LIN {X 0,Y 196.3,Z 471.05,A -85,B 0,C 180,E1 -25408.972,E2 -25408.972} C_VEL
LIN {X 0,Y 193.786,Z 486.083,A -85,B 0,C 180,E1 -25409.629,E2 -25409.629} C_VEL
LIN {X 0,Y 190.214,Z 500.774,A -85,B 0,C 180,E1 -25410.535,E2 -25410.535} C_VEL
LIN {X 0,Y 185.876,Z 514.562,A -85,B 0,C 180,E1 -25411.712,E2 -25411.712} C_VEL
LIN {X 0,Y 180.555,Z 528.47,A -85,B 0,C 180,E1 -25413.314,E2 -25413.314} C_VEL
LIN {X 0,Y 174.309,Z 541.829,A -85,B 0,C 180,E1 -25415.27,E2 -25415.27} C_VEL
LIN {X 0,Y 167.482,Z 554.228,A -85,B 0,C 180,E1 -25417.625,E2 -25417.625} C_VEL
LIN {X 0,Y 160.938,Z 564.609,A -85,B 0,C 180,E1 -25420.166,E2 -25420.166} C_VEL
LIN {X 0,Y 154.161,Z 574.239,A -85,B 0,C 180,E1 -25423.164,E2 -25423.164} C_VEL
LIN {X 0,Y 148.078,Z 582.443,A -85,B 0,C 180,E1 -25426.515,E2 -25426.515} C_VEL
LIN {X 0,Y 141.347,Z 590.516,A -85,B 0,C 180,E1 -25430.659,E2 -25430.659} C_VEL
LIN {X 0,Y 135.368,Z 597.175,A -85,B 0,C 180,E1 -25435.175,E2 -25435.175} C_VEL
LIN {X 0,Y 129.686,Z 603.328,A -85,B 0,C 180,E1 -25440.809,E2 -25440.809} C_VEL
LIN {X 0,Y 125.219,Z 608.071,A -85,B 0,C 180,E1 -25446.867,E2 -25446.867} C_VEL
LIN {X 0,Y 122.097,Z 611.536,A -85,B 0,C 180,E1 -25453.274,E2 -25453.274} C_VEL
LIN {X 0,Y 120.197,Z 613.818,A -85,B 0,C 180,E1 -25459.898,E2 -25459.898} C_VEL
LIN {X 0,Y 119.437,Z 614.974,A -85,B 0,C 180,E1 -25466.627,E2 -25466.627} C_VEL
LIN {X 0,Y 119.419,Z 615.126,A -85,B 0,C 180,E1 -25470,E2 -25470} C_VEL
LIN {X 0,Y 119.683,Z 614.566,A -85,B 0,C 180,E1 -25476.744,E2 -25476.744} C_VEL
LIN {X 0,Y 120.982,Z 612.894,A -85,B 0,C 180,E1 -25483.436,E2 -25483.436} C_VEL
LIN {X 0,Y 123.4,Z 610.069,A -85,B 0,C 180,E1 -25489.981,E2 -25489.981} C_VEL
LIN {X 0,Y 127.319,Z 606.012,A -85,B 0,C 180,E1 -25496.205,E2 -25496.205} C_VEL
LIN {X 0,Y 132.367,Z 600.63,A -85,B 0,C 180,E1 -25502.068,E2 -25502.068} C_VEL
LIN {X 0,Y 138.615,Z 593.765,A -85,B 0,C 180,E1 -25507.474,E2 -25507.474} C_VEL
LIN {X 0,Y 145.953,Z 585.189,A -85,B 0,C 180,E1 -25512.386,E2 -25512.386} C_VEL
LIN {X 0,Y 150.8,Z 579.119,A -85,B 0,C 180,E1 -25515.081,E2 -25515.081} C_VEL
LIN {X 0,Y 156.318,Z 571.624,A -85,B 0,C 180,E1 -25517.886,E2 -25517.886} C_VEL
LIN {X 0,Y 163.24,Z 561.484,A -85,B 0,C 180,E1 -25520.799,E2 -25520.799} C_VEL
LIN {X 0,Y 170.453,Z 549.406,A -85,B 0,C 180,E1 -25523.512,E2 -25523.512} C_VEL
LIN {X 0,Y 176.765,Z 537.285,A -85,B 0,C 180,E1 -25525.586,E2 -25525.586} C_VEL
LIN {X 0,Y 182.653,Z 523.835,A -85,B 0,C 180,E1 -25527.406,E2 -25527.406} C_VEL
LIN {X 0,Y 187.121,Z 511.539,A -85,B 0,C 180,E1 -25528.697,E2 -25528.697} C_VEL
LIN {X 0,Y 191.471,Z 496.805,A -85,B 0,C 180,E1 -25529.865,E2 -25529.865} C_VEL
LIN {X 0,Y 194.807,Z 481.709,A -85,B 0,C 180,E1 -25530.722,E2 -25530.722} C_VEL
LIN {X 0,Y 197.091,Z 466.466,A -85,B 0,C 180,E1 -25531.281,E2 -25531.281} C_VEL
LIN {X 0,Y 201.447,Z 418.406,A -85,B 0,C 180,E1 -25532.593,E2 -25532.593} C_VEL
LIN {X 0,Y 197.597,Z 410.359,A -85,B 0,C 180,E1 -25535.536,E2 -25535.536} C_VEL
LIN {X 0,Y 193.811,Z 403.079,A -85,B 0,C 180,E1 -25538.878,E2 -25538.878} C_VEL
LIN {X 0,Y 190.348,Z 396.957,A -85,B 0,C 180,E1 -25542.543,E2 -25542.543} C_VEL
LIN {X 0,Y 187.688,Z 392.59,A -85,B 0,C 180,E1 -25546.051,E2 -25546.051} C_VEL
LIN {X 0,Y 185.737,Z 388.987,A -85,B 0,C 180,E1 -25549.508,E2 -25549.508} C_VEL
LIN {X 0,Y 183.95,Z 386.282,A -85,B 0,C 180,E1 -25554.207,E2 -25554.207} C_VEL
LIN {X 0,Y 183.494,Z 384.314,A -85,B 0,C 180,E1 -25557.256,E2 -25557.256} C_VEL
LIN {X 0,Y 183.527,Z 384.307,A -85,B 0,C 180,E1 -25562.606,E2 -25562.606} C_VEL
LIN {X 0,Y 185.177,Z 388.442,A -85,B 0,C 180,E1 -25569.007,E2 -25569.007} C_VEL
LIN {X 0,Y 185.895,Z 389.445,A -85,B 0,C 180,E1 -25570.494,E2 -25570.494} C_VEL
LIN {X 0,Y 188.515,Z 393.956,A -85,B 0,C 180,E1 -25574.782,E2 -25574.782} C_VEL
LIN {X 0,Y 190.911,Z 398.053,A -85,B 0,C 180,E1 -25577.767,E2 -25577.767} C_VEL
LIN {X 0,Y 193.357,Z 402.379,A -85,B 0,C 180,E1 -25580.339,E2 -25580.339} C_VEL
LIN {X 0,Y 195.257,Z 406.102,A -85,B 0,C 180,E1 -25582.136,E2 -25582.136} C_VEL
LIN {X 0,Y 198.42,Z 414.111,A -85,B 0,C 180,E1 -25584.943,E2 -25584.943} C_VEL
LIN {X 0,Y 201.237,Z 421.993,A -85,B 0,C 180,E1 -25587.208,E2 -25587.208} C_VEL
LIN {X 0,Y 196.16,Z 476.141,A -85,B 0,C 180,E1 -25588.658,E2 -25588.658} C_VEL
LIN {X 0,Y 193.378,Z 491.918,A -85,B 0,C 180,E1 -25589.283,E2 -25589.283} C_VEL
LIN {X 0,Y 189.569,Z 507.14,A -85,B 0,C 180,E1 -25590.203,E2 -25590.203} C_VEL
LIN {X 0,Y 185.034,Z 520.859,A -85,B 0,C 180,E1 -25591.287,E2 -25591.287} C_VEL
LIN {X 0,Y 179.64,Z 534.306,A -85,B 0,C 180,E1 -25592.742,E2 -25592.742} C_VEL
LIN {X 0,Y 173.552,Z 547.041,A -85,B 0,C 180,E1 -25594.536,E2 -25594.536} C_VEL
LIN {X 0,Y 166.783,Z 559.341,A -85,B 0,C 180,E1 -25596.812,E2 -25596.812} C_VEL
LIN {X 0,Y 159.471,Z 570.819,A -85,B 0,C 180,E1 -25599.537,E2 -25599.537} C_VEL
LIN {X 0,Y 152.629,Z 580.487,A -85,B 0,C 180,E1 -25602.547,E2 -25602.547} C_VEL
LIN {X 0,Y 145.168,Z 590.115,A -85,B 0,C 180,E1 -25606.477,E2 -25606.477} C_VEL
LIN {X 0,Y 138.116,Z 598.719,A -85,B 0,C 180,E1 -25611.243,E2 -25611.243} C_VEL
LIN {X 0,Y 132.184,Z 605.322,A -85,B 0,C 180,E1 -25616.065,E2 -25616.065} C_VEL
LIN {X 0,Y 126.669,Z 611.479,A -85,B 0,C 180,E1 -25622.252,E2 -25622.252} C_VEL
LIN {X 0,Y 124.332,Z 613.407,A -85,B 0,C 180,E1 -25624.578,E2 -25624.578} C_VEL
LIN {X 0,Y 119.213,Z 616.082,A -85,B 0,C 180,E1 -25628.377,E2 -25628.377} C_VEL
LIN {X 0,Y 115.378,Z 617.848,A -85,B 0,C 180,E1 -25631.671,E2 -25631.671} C_VEL
LIN {X 0,Y 113.504,Z 618.991,A -85,B 0,C 180,E1 -25634.42,E2 -25634.42} C_VEL
LIN {X 0,Y 113.194,Z 619.293,A -85,B 0,C 180,E1 -25635.386,E2 -25635.386} C_VEL
LIN {X 0,Y 112.135,Z 621.139,A -85,B 0,C 180,E1 -25642.799,E2 -25642.799} C_VEL
LIN {X 0,Y 112.248,Z 621.75,A -85,B 0,C 180,E1 -25650,E2 -25650} C_VEL
LIN {X 0,Y 112.127,Z 621.12,A -85,B 0,C 180,E1 -25657.201,E2 -25657.201} C_VEL
LIN {X 0,Y 113.113,Z 619.332,A -85,B 0,C 180,E1 -25664.39,E2 -25664.39} C_VEL
LIN {X 0,Y 115.543,Z 616.373,A -85,B 0,C 180,E1 -25671.404,E2 -25671.404} C_VEL
LIN {X 0,Y 119.342,Z 612.172,A -85,B 0,C 180,E1 -25678.106,E2 -25678.106} C_VEL
LIN {X 0,Y 124.758,Z 606.631,A -85,B 0,C 180,E1 -25684.285,E2 -25684.285} C_VEL
LIN {X 0,Y 131.502,Z 599.596,A -85,B 0,C 180,E1 -25689.89,E2 -25689.89} C_VEL
LIN {X 0,Y 138.345,Z 591.848,A -85,B 0,C 180,E1 -25694.499,E2 -25694.499} C_VEL
LIN {X 0,Y 145.593,Z 583.013,A -85,B 0,C 180,E1 -25698.433,E2 -25698.433} C_VEL
LIN {X 0,Y 153.801,Z 572.132,A -85,B 0,C 180,E1 -25702.02,E2 -25702.02} C_VEL
LIN {X 0,Y 161.305,Z 560.935,A -85,B 0,C 180,E1 -25704.777,E2 -25704.777} C_VEL
LIN {X 0,Y 168.449,Z 548.675,A -85,B 0,C 180,E1 -25707.096,E2 -25707.096} C_VEL
LIN {X 0,Y 175.181,Z 535.171,A -85,B 0,C 180,E1 -25709.038,E2 -25709.038} C_VEL
LIN {X 0,Y 180.74,Z 521.912,A -85,B 0,C 180,E1 -25710.46,E2 -25710.46} C_VEL
LIN {X 0,Y 185.715,Z 507.4,A -85,B 0,C 180,E1 -25711.621,E2 -25711.621} C_VEL
LIN {X 0,Y 189.648,Z 492.344,A -85,B 0,C 180,E1 -25712.505,E2 -25712.505} C_VEL
LIN {X 0,Y 192.467,Z 477.05,A -85,B 0,C 180,E1 -25713.108,E2 -25713.108} C_VEL
LIN {X 0,Y 195.922,Z 442.724,A -85,B 0,C 180,E1 -25714.03,E2 -25714.03} C_VEL
LIN {X 0,Y 197.57,Z 424.787,A -85,B 0,C 180,E1 -25714.509,E2 -25714.509} C_VEL
LIN {X 0,Y 194.282,Z 415.387,A -85,B 0,C 180,E1 -25717.467,E2 -25717.467} C_VEL
LIN {X 0,Y 191.942,Z 409.582,A -85,B 0,C 180,E1 -25719.796,E2 -25719.796} C_VEL
LIN {X 0,Y 188.507,Z 403.239,A -85,B 0,C 180,E1 -25723.624,E2 -25723.624} C_VEL
LIN {X 0,Y 186.244,Z 399.273,A -85,B 0,C 180,E1 -25726.776,E2 -25726.776} C_VEL
LIN {X 0,Y 184.295,Z 395.581,A -85,B 0,C 180,E1 -25730.396,E2 -25730.396} C_VEL
LIN {X 0,Y 182.635,Z 392.54,A -85,B 0,C 180,E1 -25735.31,E2 -25735.31} C_VEL
LIN {X 0,Y 182.364,Z 391.3,A -85,B 0,C 180,E1 -25737.239,E2 -25737.239} C_VEL
LIN {X 0,Y 182.151,Z 391.03,A -85,B 0,C 180,E1 -25740,E2 -25740} C_VEL
LIN {X 0,Y 182.429,Z 391.531,A -85,B 0,C 180,E1 -25743.728,E2 -25743.728} C_VEL
LIN {X 0,Y 183.828,Z 395.187,A -85,B 0,C 180,E1 -25749.074,E2 -25749.074} C_VEL
LIN {X 0,Y 184.521,Z 396.112,A -85,B 0,C 180,E1 -25750.562,E2 -25750.562} C_VEL
LIN {X 0,Y 186.923,Z 400.501,A -85,B 0,C 180,E1 -25754.702,E2 -25754.702} C_VEL
LIN {X 0,Y 189.266,Z 404.677,A -85,B 0,C 180,E1 -25757.756,E2 -25757.756} C_VEL
LIN {X 0,Y 192.494,Z 410.713,A -85,B 0,C 180,E1 -25761.204,E2 -25761.204} C_VEL
LIN {X 0,Y 195.769,Z 417.37,A -85,B 0,C 180,E1 -25764.172,E2 -25764.172} C_VEL
LIN {X 0,Y 197.776,Z 421.755,A -85,B 0,C 180,E1 -25765.813,E2 -25765.813} C_VEL
LIN {X 0,Y 193.089,Z 470.398,A -85,B 0,C 180,E1 -25767.1,E2 -25767.1} C_VEL
LIN {X 0,Y 190.382,Z 486.296,A -85,B 0,C 180,E1 -25767.775,E2 -25767.775} C_VEL
LIN {X 0,Y 186.708,Z 500.985,A -85,B 0,C 180,E1 -25768.658,E2 -25768.658} C_VEL
LIN {X 0,Y 182.243,Z 514.772,A -85,B 0,C 180,E1 -25769.812,E2 -25769.812} C_VEL
LIN {X 0,Y 176.917,Z 528.235,A -85,B 0,C 180,E1 -25771.322,E2 -25771.322} C_VEL
LIN {X 0,Y 170.981,Z 540.748,A -85,B 0,C 180,E1 -25773.126,E2 -25773.126} C_VEL
LIN {X 0,Y 164.496,Z 552.307,A -85,B 0,C 180,E1 -25775.207,E2 -25775.207} C_VEL
LIN {X 0,Y 157.704,Z 563.04,A -85,B 0,C 180,E1 -25777.721,E2 -25777.721} C_VEL
LIN {X 0,Y 150.543,Z 572.967,A -85,B 0,C 180,E1 -25780.659,E2 -25780.659} C_VEL
LIN {X 0,Y 143.006,Z 582.648,A -85,B 0,C 180,E1 -25784.555,E2 -25784.555} C_VEL
LIN {X 0,Y 135.9,Z 590.722,A -85,B 0,C 180,E1 -25788.75,E2 -25788.75} C_VEL
LIN {X 0,Y 129.57,Z 597.381,A -85,B 0,C 180,E1 -25793.371,E2 -25793.371} C_VEL
LIN {X 0,Y 123.508,Z 603.533,A -85,B 0,C 180,E1 -25799.195,E2 -25799.195} C_VEL
LIN {X 0,Y 118.713,Z 608.276,A -85,B 0,C 180,E1 -25805.518,E2 -25805.518} C_VEL
LIN {X 0,Y 115.272,Z 611.741,A -85,B 0,C 180,E1 -25812.252,E2 -25812.252} C_VEL
LIN {X 0,Y 113.203,Z 614.022,A -85,B 0,C 180,E1 -25819.266,E2 -25819.266} C_VEL
LIN {X 0,Y 112.353,Z 615.177,A -85,B 0,C 180,E1 -25826.414,E2 -25826.414} C_VEL
LIN {X 0,Y 112.335,Z 615.329,A -85,B 0,C 180,E1 -25830,E2 -25830} C_VEL
LIN {X 0,Y 112.624,Z 614.769,A -85,B 0,C 180,E1 -25837.169,E2 -25837.169} C_VEL
LIN {X 0,Y 114.05,Z 613.098,A -85,B 0,C 180,E1 -25844.269,E2 -25844.269} C_VEL
LIN {X 0,Y 116.717,Z 610.273,A -85,B 0,C 180,E1 -25851.178,E2 -25851.178} C_VEL
LIN {X 0,Y 120.945,Z 606.215,A -85,B 0,C 180,E1 -25857.701,E2 -25857.701} C_VEL
LIN {X 0,Y 126.368,Z 600.833,A -85,B 0,C 180,E1 -25863.789,E2 -25863.789} C_VEL
LIN {X 0,Y 133.009,Z 593.968,A -85,B 0,C 180,E1 -25869.349,E2 -25869.349} C_VEL
LIN {X 0,Y 140.792,Z 585.39,A -85,B 0,C 180,E1 -25874.333,E2 -25874.333} C_VEL
LIN {X 0,Y 146.284,Z 578.73,A -85,B 0,C 180,E1 -25877.329,E2 -25877.329} C_VEL
LIN {X 0,Y 152.796,Z 570.211,A -85,B 0,C 180,E1 -25880.391,E2 -25880.391} C_VEL
LIN {X 0,Y 160.079,Z 559.807,A -85,B 0,C 180,E1 -25883.246,E2 -25883.246} C_VEL
LIN {X 0,Y 166.963,Z 548.488,A -85,B 0,C 180,E1 -25885.695,E2 -25885.695} C_VEL
LIN {X 0,Y 173.517,Z 536.181,A -85,B 0,C 180,E1 -25887.724,E2 -25887.724} C_VEL
LIN {X 0,Y 179.503,Z 522.719,A -85,B 0,C 180,E1 -25889.467,E2 -25889.467} C_VEL
LIN {X 0,Y 184.555,Z 508.759,A -85,B 0,C 180,E1 -25890.862,E2 -25890.862} C_VEL
LIN {X 0,Y 188.693,Z 494.404,A -85,B 0,C 180,E1 -25891.913,E2 -25891.913} C_VEL
LIN {X 0,Y 192.06,Z 478.698,A -85,B 0,C 180,E1 -25892.714,E2 -25892.714} C_VEL
LIN {X 0,Y 194.184,Z 463.277,A -85,B 0,C 180,E1 -25893.208,E2 -25893.208} C_VEL
LIN {X 0,Y 198.031,Z 421.974,A -85,B 0,C 180,E1 -25894.285,E2 -25894.285} C_VEL
LIN {X 0,Y 194.199,Z 413.869,A -85,B 0,C 180,E1 -25897.526,E2 -25897.526} C_VEL
LIN {X 0,Y 190.907,Z 407.427,A -85,B 0,C 180,E1 -25900.79,E2 -25900.79} C_VEL
LIN {X 0,Y 188.19,Z 402.537,A -85,B 0,C 180,E1 -25904.013,E2 -25904.013} C_VEL
LIN {X 0,Y 186.384,Z 399.332,A -85,B 0,C 180,E1 -25906.63,E2 -25906.63} C_VEL
LIN {X 0,Y 184.403,Z 395.666,A -85,B 0,C 180,E1 -25910.401,E2 -25910.401} C_VEL
LIN {X 0,Y 182.769,Z 392.393,A -85,B 0,C 180,E1 -25915.796,E2 -25915.796} C_VEL
LIN {X 0,Y 182.625,Z 391.396,A -85,B 0,C 180,E1 -25917.243,E2 -25917.243} C_VEL
LIN {X 0,Y 182.608,Z 391.312,A -85,B 0,C 180,E1 -25922.205,E2 -25922.205} C_VEL
LIN {X 0,Y 184.439,Z 395.708,A -85,B 0,C 180,E1 -25929.32,E2 -25929.32} C_VEL
LIN {X 0,Y 187.113,Z 400.621,A -85,B 0,C 180,E1 -25934.131,E2 -25934.131} C_VEL
LIN {X 0,Y 189.335,Z 404.558,A -85,B 0,C 180,E1 -25937.066,E2 -25937.066} C_VEL
LIN {X 0,Y 192.506,Z 410.448,A -85,B 0,C 180,E1 -25940.502,E2 -25940.502} C_VEL
LIN {X 0,Y 195.434,Z 418.137,A -85,B 0,C 180,E1 -25943.371,E2 -25943.371} C_VEL
LIN {X 0,Y 197.796,Z 425.06,A -85,B 0,C 180,E1 -25945.469,E2 -25945.469} C_VEL
LIN {X 0,Y 192.822,Z 476.142,A -85,B 0,C 180,E1 -25946.81,E2 -25946.81} C_VEL
LIN {X 0,Y 190.008,Z 491.724,A -85,B 0,C 180,E1 -25947.416,E2 -25947.416} C_VEL
LIN {X 0,Y 186.079,Z 506.942,A -85,B 0,C 180,E1 -25948.302,E2 -25948.302} C_VEL
LIN {X 0,Y 181.444,Z 520.662,A -85,B 0,C 180,E1 -25949.368,E2 -25949.368} C_VEL
LIN {X 0,Y 175.9,Z 534.108,A -85,B 0,C 180,E1 -25950.796,E2 -25950.796} C_VEL
LIN {X 0,Y 169.641,Z 546.794,A -85,B 0,C 180,E1 -25952.547,E2 -25952.547} C_VEL
LIN {X 0,Y 162.618,Z 559.141,A -85,B 0,C 180,E1 -25954.803,E2 -25954.803} C_VEL
LIN {X 0,Y 155.01,Z 570.617,A -85,B 0,C 180,E1 -25957.495,E2 -25957.495} C_VEL
LIN {X 0,Y 147.888,Z 580.285,A -85,B 0,C 180,E1 -25960.506,E2 -25960.506} C_VEL
LIN {X 0,Y 140.157,Z 589.787,A -85,B 0,C 180,E1 -25964.396,E2 -25964.396} C_VEL
LIN {X 0,Y 133.324,Z 597.716,A -85,B 0,C 180,E1 -25968.784,E2 -25968.784} C_VEL
LIN {X 0,Y 126.283,Z 605.118,A -85,B 0,C 180,E1 -25974.244,E2 -25974.244} C_VEL
LIN {X 0,Y 120.625,Z 611.002,A -85,B 0,C 180,E1 -25980.315,E2 -25980.315} C_VEL
LIN {X 0,Y 117.351,Z 614.51,A -85,B 0,C 180,E1 -25985.215,E2 -25985.215} C_VEL
LIN {X 0,Y 114.117,Z 618.057,A -85,B 0,C 180,E1 -25992.066,E2 -25992.066} C_VEL
LIN {X 0,Y 113.194,Z 619.293,A -85,B 0,C 180,E1 -25995.386,E2 -25995.386} C_VEL
LIN {X 0,Y 112.042,Z 620.233,A -85,B 0,C 180,E1 -25998.29,E2 -25998.29} C_VEL
LIN {X 0,Y 110.209,Z 620.902,A -85,B 0,C 180,E1 -26001.18,E2 -26001.18} C_VEL
LIN {X 0,Y 106.313,Z 621.518,A -85,B 0,C 180,E1 -26007.182,E2 -26007.182} C_VEL
LIN {X 0,Y 105.049,Z 621.484,A -85,B 0,C 180,E1 -26011.468,E2 -26011.468} C_VEL
LIN {X 0,Y 105.054,Z 620.915,A -85,B 0,C 180,E1 -26017.689,E2 -26017.689} C_VEL
LIN {X 0,Y 106.195,Z 619.127,A -85,B 0,C 180,E1 -26025.35,E2 -26025.35} C_VEL
LIN {X 0,Y 108.882,Z 616.167,A -85,B 0,C 180,E1 -26032.785,E2 -26032.785} C_VEL
LIN {X 0,Y 113.068,Z 611.966,A -85,B 0,C 180,E1 -26039.818,E2 -26039.818} C_VEL
LIN {X 0,Y 118.897,Z 606.424,A -85,B 0,C 180,E1 -26046.234,E2 -26046.234} C_VEL
LIN {X 0,Y 126.073,Z 599.389,A -85,B 0,C 180,E1 -26051.984,E2 -26051.984} C_VEL
LIN {X 0,Y 134.165,Z 590.637,A -85,B 0,C 180,E1 -26057.168,E2 -26057.168} C_VEL
LIN {X 0,Y 142.145,Z 581.353,A -85,B 0,C 180,E1 -26061.141,E2 -26061.141} C_VEL
LIN {X 0,Y 149.5,Z 571.924,A -85,B 0,C 180,E1 -26064.184,E2 -26064.184} C_VEL
LIN {X 0,Y 157.306,Z 560.729,A -85,B 0,C 180,E1 -26066.895,E2 -26066.895} C_VEL
LIN {X 0,Y 164.799,Z 548.256,A -85,B 0,C 180,E1 -26069.22,E2 -26069.22} C_VEL
LIN {X 0,Y 171.632,Z 534.963,A -85,B 0,C 180,E1 -26071.074,E2 -26071.074} C_VEL
LIN {X 0,Y 177.35,Z 521.704,A -85,B 0,C 180,E1 -26072.455,E2 -26072.455} C_VEL
LIN {X 0,Y 182.449,Z 507.19,A -85,B 0,C 180,E1 -26073.582,E2 -26073.582} C_VEL
LIN {X 0,Y 186.479,Z 492.131,A -85,B 0,C 180,E1 -26074.439,E2 -26074.439} C_VEL
LIN {X 0,Y 189.288,Z 477.3,A -85,B 0,C 180,E1 -26075.008,E2 -26075.008} C_VEL
LIN {X 0,Y 192.26,Z 449.441,A -85,B 0,C 180,E1 -26075.744,E2 -26075.744} C_VEL
LIN {X 0,Y 194.297,Z 427.907,A -85,B 0,C 180,E1 -26076.313,E2 -26076.313} C_VEL
LIN {X 0,Y 191.509,Z 419.557,A -85,B 0,C 180,E1 -26079.105,E2 -26079.105} C_VEL
LIN {X 0,Y 189.918,Z 415.545,A -85,B 0,C 180,E1 -26080.827,E2 -26080.827} C_VEL
LIN {X 0,Y 186.997,Z 409.783,A -85,B 0,C 180,E1 -26084.328,E2 -26084.328} C_VEL
LIN {X 0,Y 184.859,Z 405.856,A -85,B 0,C 180,E1 -26087.513,E2 -26087.513} C_VEL
LIN {X 0,Y 183.045,Z 402.324,A -85,B 0,C 180,E1 -26091.166,E2 -26091.166} C_VEL
LIN {X 0,Y 181.513,Z 398.523,A -85,B 0,C 180,E1 -26097.018,E2 -26097.018} C_VEL
LIN {X 0,Y 181.285,Z 398.078,A -85,B 0,C 180,E1 -26100,E2 -26100} C_VEL
LIN {X 0,Y 181.503,Z 398.469,A -85,B 0,C 180,E1 -26103.33,E2 -26103.33} C_VEL
LIN {X 0,Y 182.735,Z 402.024,A -85,B 0,C 180,E1 -26108.571,E2 -26108.571} C_VEL
LIN {X 0,Y 183.447,Z 403.081,A -85,B 0,C 180,E1 -26110.206,E2 -26110.206} C_VEL
LIN {X 0,Y 185.671,Z 407.394,A -85,B 0,C 180,E1 -26114.243,E2 -26114.243} C_VEL
LIN {X 0,Y 187.833,Z 411.455,A -85,B 0,C 180,E1 -26117.207,E2 -26117.207} C_VEL
LIN {X 0,Y 191.052,Z 417.854,A -85,B 0,C 180,E1 -26120.807,E2 -26120.807} C_VEL
LIN {X 0,Y 193.879,Z 424.017,A -85,B 0,C 180,E1 -26123.5,E2 -26123.5} C_VEL
LIN {X 0,Y 194.477,Z 425.359,A -85,B 0,C 180,E1 -26124.027,E2 -26124.027} C_VEL
LIN {X 0,Y 189.877,Z 471.308,A -85,B 0,C 180,E1 -26125.226,E2 -26125.226} C_VEL
LIN {X 0,Y 187.181,Z 486.509,A -85,B 0,C 180,E1 -26125.853,E2 -26125.853} C_VEL
LIN {X 0,Y 183.418,Z 501.195,A -85,B 0,C 180,E1 -26126.717,E2 -26126.717} C_VEL
LIN {X 0,Y 178.818,Z 514.981,A -85,B 0,C 180,E1 -26127.837,E2 -26127.837} C_VEL
LIN {X 0,Y 173.1,Z 528.968,A -85,B 0,C 180,E1 -26129.378,E2 -26129.378} C_VEL
LIN {X 0,Y 166.527,Z 542.242,A -85,B 0,C 180,E1 -26131.285,E2 -26131.285} C_VEL
LIN {X 0,Y 159.205,Z 554.641,A -85,B 0,C 180,E1 -26133.571,E2 -26133.571} C_VEL
LIN {X 0,Y 152.165,Z 565.021,A -85,B 0,C 180,E1 -26136.075,E2 -26136.075} C_VEL
LIN {X 0,Y 144.085,Z 575.518,A -85,B 0,C 180,E1 -26139.353,E2 -26139.353} C_VEL
LIN {X 0,Y 136.98,Z 584.077,A -85,B 0,C 180,E1 -26143.021,E2 -26143.021} C_VEL
LIN {X 0,Y 129.619,Z 591.927,A -85,B 0,C 180,E1 -26147.333,E2 -26147.333} C_VEL
LIN {X 0,Y 122.174,Z 599.251,A -85,B 0,C 180,E1 -26152.844,E2 -26152.844} C_VEL
LIN {X 0,Y 115.996,Z 605.051,A -85,B 0,C 180,E1 -26159.003,E2 -26159.003} C_VEL
LIN {X 0,Y 112.276,Z 608.48,A -85,B 0,C 180,E1 -26164.014,E2 -26164.014} C_VEL
LIN {X 0,Y 108.494,Z 611.945,A -85,B 0,C 180,E1 -26171.102,E2 -26171.102} C_VEL
LIN {X 0,Y 106.216,Z 614.226,A -85,B 0,C 180,E1 -26178.551,E2 -26178.551} C_VEL
LIN {X 0,Y 105.265,Z 615.38,A -85,B 0,C 180,E1 -26186.172,E2 -26186.172} C_VEL
LIN {X 0,Y 105.237,Z 615.532,A -85,B 0,C 180,E1 -26190,E2 -26190} C_VEL
LIN {X 0,Y 105.592,Z 614.972,A -85,B 0,C 180,E1 -26197.649,E2 -26197.649} C_VEL
LIN {X 0,Y 107.157,Z 613.301,A -85,B 0,C 180,E1 -26205.209,E2 -26205.209} C_VEL
LIN {X 0,Y 110.093,Z 610.476,A -85,B 0,C 180,E1 -26212.52,E2 -26212.52} C_VEL
LIN {X 0,Y 114.654,Z 606.419,A -85,B 0,C 180,E1 -26219.365,E2 -26219.365} C_VEL
LIN {X 0,Y 120.496,Z 601.036,A -85,B 0,C 180,E1 -26225.679,E2 -26225.679} C_VEL
LIN {X 0,Y 127.579,Z 594.17,A -85,B 0,C 180,E1 -26231.379,E2 -26231.379} C_VEL
LIN {X 0,Y 134.676,Z 586.787,A -85,B 0,C 180,E1 -26235.85,E2 -26235.85} C_VEL
LIN {X 0,Y 140.198,Z 580.569,A -85,B 0,C 180,E1 -26238.756,E2 -26238.756} C_VEL
LIN {X 0,Y 145.939,Z 573.518,A -85,B 0,C 180,E1 -26241.493,E2 -26241.493} C_VEL
LIN {X 0,Y 153.364,Z 563.66,A -85,B 0,C 180,E1 -26244.428,E2 -26244.428} C_VEL
LIN {X 0,Y 161.08,Z 551.935,A -85,B 0,C 180,E1 -26247.126,E2 -26247.126} C_VEL
LIN {X 0,Y 168.464,Z 538.969,A -85,B 0,C 180,E1 -26249.363,E2 -26249.363} C_VEL
LIN {X 0,Y 174.776,Z 525.676,A -85,B 0,C 180,E1 -26251.148,E2 -26251.148} C_VEL
LIN {X 0,Y 180.165,Z 511.931,A -85,B 0,C 180,E1 -26252.551,E2 -26252.551} C_VEL
LIN {X 0,Y 184.765,Z 497.193,A -85,B 0,C 180,E1 -26253.667,E2 -26253.667} C_VEL
LIN {X 0,Y 188.185,Z 482.602,A -85,B 0,C 180,E1 -26254.461,E2 -26254.461} C_VEL
LIN {X 0,Y 190.589,Z 467.616,A -85,B 0,C 180,E1 -26254.999,E2 -26254.999} C_VEL
LIN {X 0,Y 194.71,Z 425.601,A -85,B 0,C 180,E1 -26256.086,E2 -26256.086} C_VEL
LIN {X 0,Y 191.488,Z 418.43,A -85,B 0,C 180,E1 -26259.116,E2 -26259.116} C_VEL
LIN {X 0,Y 188.418,Z 412.32,A -85,B 0,C 180,E1 -26262.498,E2 -26262.498} C_VEL
LIN {X 0,Y 186.278,Z 408.315,A -85,B 0,C 180,E1 -26265.344,E2 -26265.344} C_VEL
LIN {X 0,Y 185.082,Z 406.027,A -85,B 0,C 180,E1 -26267.249,E2 -26267.249} C_VEL
LIN {X 0,Y 183.291,Z 402.526,A -85,B 0,C 180,E1 -26270.899,E2 -26270.899} C_VEL
LIN {X 0,Y 181.794,Z 399.091,A -85,B 0,C 180,E1 -26276.537,E2 -26276.537} C_VEL
LIN {X 0,Y 181.701,Z 398.351,A -85,B 0,C 180,E1 -26277.783,E2 -26277.783} C_VEL
LIN {X 0,Y 181.737,Z 398.416,A -85,B 0,C 180,E1 -26282.216,E2 -26282.216} C_VEL
LIN {X 0,Y 183.207,Z 402.429,A -85,B 0,C 180,E1 -26288.548,E2 -26288.548} C_VEL
LIN {X 0,Y 183.785,Z 403.582,A -85,B 0,C 180,E1 -26289.909,E2 -26289.909} C_VEL
LIN {X 0,Y 185.779,Z 407.347,A -85,B 0,C 180,E1 -26293.537,E2 -26293.537} C_VEL
LIN {X 0,Y 188.053,Z 411.631,A -85,B 0,C 180,E1 -26296.696,E2 -26296.696} C_VEL
LIN {X 0,Y 190.757,Z 417.016,A -85,B 0,C 180,E1 -26299.785,E2 -26299.785} C_VEL
LIN {X 0,Y 193.452,Z 424.761,A -85,B 0,C 180,E1 -26302.616,E2 -26302.616} C_VEL
LIN {X 0,Y 194.519,Z 428.093,A -85,B 0,C 180,E1 -26303.653,E2 -26303.653} C_VEL
LIN {X 0,Y 189.702,Z 476.124,A -85,B 0,C 180,E1 -26304.905,E2 -26304.905} C_VEL
LIN {X 0,Y 186.847,Z 491.531,A -85,B 0,C 180,E1 -26305.484,E2 -26305.484} C_VEL
LIN {X 0,Y 182.811,Z 506.746,A -85,B 0,C 180,E1 -26306.336,E2 -26306.336} C_VEL
LIN {X 0,Y 178.07,Z 520.465,A -85,B 0,C 180,E1 -26307.377,E2 -26307.377} C_VEL
LIN {X 0,Y 172.36,Z 533.909,A -85,B 0,C 180,E1 -26308.76,E2 -26308.76} C_VEL
LIN {X 0,Y 166.058,Z 546.316,A -85,B 0,C 180,E1 -26310.427,E2 -26310.427} C_VEL
LIN {X 0,Y 158.667,Z 558.941,A -85,B 0,C 180,E1 -26312.694,E2 -26312.694} C_VEL
LIN {X 0,Y 150.766,Z 570.416,A -85,B 0,C 180,E1 -26315.339,E2 -26315.339} C_VEL
LIN {X 0,Y 143.336,Z 580.082,A -85,B 0,C 180,E1 -26318.327,E2 -26318.327} C_VEL
LIN {X 0,Y 135.229,Z 589.583,A -85,B 0,C 180,E1 -26322.22,E2 -26322.22} C_VEL
LIN {X 0,Y 128.006,Z 597.512,A -85,B 0,C 180,E1 -26326.664,E2 -26326.664} C_VEL
LIN {X 0,Y 120.537,Z 604.914,A -85,B 0,C 180,E1 -26332.252,E2 -26332.252} C_VEL
LIN {X 0,Y 114.45,Z 610.798,A -85,B 0,C 180,E1 -26338.537,E2 -26338.537} C_VEL
LIN {X 0,Y 110.886,Z 614.306,A -85,B 0,C 180,E1 -26343.663,E2 -26343.663} C_VEL
LIN {X 0,Y 107.331,Z 617.853,A -85,B 0,C 180,E1 -26350.89,E2 -26350.89} C_VEL
LIN {X 0,Y 105.484,Z 620.199,A -85,B 0,C 180,E1 -26358.47,E2 -26358.47} C_VEL
LIN {X 0,Y 105.007,Z 621.387,A -85,B 0,C 180,E1 -26366.162,E2 -26366.162} C_VEL
LIN {X 0,Y 105.166,Z 621.548,A -85,B 0,C 180,E1 -26370,E2 -26370} C_VEL
LIN {X 0,Y 105.049,Z 621.484,A -85,B 0,C 180,E1 -26371.468,E2 -26371.468} C_VEL
LIN {X 0,Y 104.287,Z 621.291,A -85,B 0,C 180,E1 -26374.668,E2 -26374.668} C_VEL
LIN {X 0,Y 101.684,Z 620.469,A -85,B 0,C 180,E1 -26379.978,E2 -26379.978} C_VEL
LIN {X 0,Y 99.934,Z 619.491,A -85,B 0,C 180,E1 -26384.385,E2 -26384.385} C_VEL
LIN {X 0,Y 99.851,Z 618.377,A -85,B 0,C 180,E1 -26388.319,E2 -26388.319} C_VEL
LIN {X 0,Y 100.01,Z 618.119,A -85,B 0,C 180,E1 -26388.872,E2 -26388.872} C_VEL
LIN {X 0,Y 102.292,Z 615.96,A -85,B 0,C 180,E1 -26394.344,E2 -26394.344} C_VEL
LIN {X 0,Y 106.92,Z 611.761,A -85,B 0,C 180,E1 -26401.725,E2 -26401.725} C_VEL
LIN {X 0,Y 113.18,Z 606.218,A -85,B 0,C 180,E1 -26408.385,E2 -26408.385} C_VEL
LIN {X 0,Y 120.843,Z 599.182,A -85,B 0,C 180,E1 -26414.257,E2 -26414.257} C_VEL
LIN {X 0,Y 128.298,Z 591.623,A -85,B 0,C 180,E1 -26418.903,E2 -26418.903} C_VEL
LIN {X 0,Y 136.523,Z 582.599,A -85,B 0,C 180,E1 -26422.929,E2 -26422.929} C_VEL
LIN {X 0,Y 145.435,Z 571.717,A -85,B 0,C 180,E1 -26426.467,E2 -26426.467} C_VEL
LIN {X 0,Y 153.535,Z 560.522,A -85,B 0,C 180,E1 -26429.12,E2 -26429.12} C_VEL
LIN {X 0,Y 160.724,Z 548.951,A -85,B 0,C 180,E1 -26431.25,E2 -26431.25} C_VEL
LIN {X 0,Y 167.578,Z 536.186,A -85,B 0,C 180,E1 -26433.021,E2 -26433.021} C_VEL
LIN {X 0,Y 173.436,Z 523.264,A -85,B 0,C 180,E1 -26434.368,E2 -26434.368} C_VEL
LIN {X 0,Y 178.638,Z 509.238,A -85,B 0,C 180,E1 -26435.472,E2 -26435.472} C_VEL
LIN {X 0,Y 182.957,Z 494.207,A -85,B 0,C 180,E1 -26436.333,E2 -26436.333} C_VEL
LIN {X 0,Y 186.096,Z 478.965,A -85,B 0,C 180,E1 -26436.922,E2 -26436.922} C_VEL
LIN {X 0,Y 188.504,Z 458.616,A -85,B 0,C 180,E1 -26437.483,E2 -26437.483} C_VEL
LIN {X 0,Y 191.212,Z 431.099,A -85,B 0,C 180,E1 -26438.176,E2 -26438.176} C_VEL
LIN {X 0,Y 188.943,Z 423.955,A -85,B 0,C 180,E1 -26440.724,E2 -26440.724} C_VEL
LIN {X 0,Y 187.789,Z 421.09,A -85,B 0,C 180,E1 -26442.086,E2 -26442.086} C_VEL
LIN {X 0,Y 185.232,Z 415.854,A -85,B 0,C 180,E1 -26445.442,E2 -26445.442} C_VEL
LIN {X 0,Y 183.543,Z 412.509,A -85,B 0,C 180,E1 -26448.193,E2 -26448.193} C_VEL
LIN {X 0,Y 181.945,Z 409.173,A -85,B 0,C 180,E1 -26451.672,E2 -26451.672} C_VEL
LIN {X 0,Y 180.564,Z 405.29,A -85,B 0,C 180,E1 -26457.77,E2 -26457.77} C_VEL
LIN {X 0,Y 180.511,Z 405.276,A -85,B 0,C 180,E1 -26462.232,E2 -26462.232} C_VEL
LIN {X 0,Y 180.639,Z 405.925,A -85,B 0,C 180,E1 -26463.625,E2 -26463.625} C_VEL
LIN {X 0,Y 181.987,Z 409.264,A -85,B 0,C 180,E1 -26468.886,E2 -26468.886} C_VEL
LIN {X 0,Y 184.19,Z 413.757,A -85,B 0,C 180,E1 -26473.375,E2 -26473.375} C_VEL
LIN {X 0,Y 186.26,Z 417.896,A -85,B 0,C 180,E1 -26476.439,E2 -26476.439} C_VEL
LIN {X 0,Y 189.168,Z 424.048,A -85,B 0,C 180,E1 -26479.924,E2 -26479.924} C_VEL
LIN {X 0,Y 191.344,Z 429.064,A -85,B 0,C 180,E1 -26482.169,E2 -26482.169} C_VEL
LIN {X 0,Y 186.895,Z 471.959,A -85,B 0,C 180,E1 -26483.275,E2 -26483.275} C_VEL
LIN {X 0,Y 184.205,Z 486.721,A -85,B 0,C 180,E1 -26483.871,E2 -26483.871} C_VEL
LIN {X 0,Y 180.346,Z 501.405,A -85,B 0,C 180,E1 -26484.708,E2 -26484.708} C_VEL
LIN {X 0,Y 175.623,Z 515.19,A -85,B 0,C 180,E1 -26485.793,E2 -26485.793} C_VEL
LIN {X 0,Y 169.531,Z 529.622,A -85,B 0,C 180,E1 -26487.342,E2 -26487.342} C_VEL
LIN {X 0,Y 162.958,Z 542.449,A -85,B 0,C 180,E1 -26489.155,E2 -26489.155} C_VEL
LIN {X 0,Y 155.389,Z 554.848,A -85,B 0,C 180,E1 -26491.388,E2 -26491.388} C_VEL
LIN {X 0,Y 148.1,Z 565.227,A -85,B 0,C 180,E1 -26493.857,E2 -26493.857} C_VEL
LIN {X 0,Y 140.422,Z 574.856,A -85,B 0,C 180,E1 -26496.797,E2 -26496.797} C_VEL
LIN {X 0,Y 132.236,Z 584.282,A -85,B 0,C 180,E1 -26500.771,E2 -26500.771} C_VEL
LIN {X 0,Y 124.463,Z 592.133,A -85,B 0,C 180,E1 -26505.105,E2 -26505.105} C_VEL
LIN {X 0,Y 116.563,Z 599.456,A -85,B 0,C 180,E1 -26510.724,E2 -26510.724} C_VEL
LIN {X 0,Y 109.942,Z 605.256,A -85,B 0,C 180,E1 -26517.088,E2 -26517.088} C_VEL
LIN {X 0,Y 105.91,Z 608.685,A -85,B 0,C 180,E1 -26522.323,E2 -26522.323} C_VEL
LIN {X 0,Y 101.774,Z 612.15,A -85,B 0,C 180,E1 -26529.802,E2 -26529.802} C_VEL
LIN {X 0,Y 99.262,Z 614.429,A -85,B 0,C 180,E1 -26537.737,E2 -26537.737} C_VEL
LIN {X 0,Y 98.189,Z 615.583,A -85,B 0,C 180,E1 -26545.896,E2 -26545.896} C_VEL
LIN {X 0,Y 98.151,Z 615.734,A -85,B 0,C 180,E1 -26550,E2 -26550} C_VEL
LIN {X 0,Y 98.553,Z 615.175,A -85,B 0,C 180,E1 -26558.2,E2 -26558.2} C_VEL
LIN {X 0,Y 100.306,Z 613.504,A -85,B 0,C 180,E1 -26566.275,E2 -26566.275} C_VEL
LIN {X 0,Y 103.539,Z 610.679,A -85,B 0,C 180,E1 -26574.032,E2 -26574.032} C_VEL
LIN {X 0,Y 108.475,Z 606.622,A -85,B 0,C 180,E1 -26581.218,E2 -26581.218} C_VEL
LIN {X 0,Y 114.772,Z 601.239,A -85,B 0,C 180,E1 -26587.758,E2 -26587.758} C_VEL
LIN {X 0,Y 122.319,Z 594.373,A -85,B 0,C 180,E1 -26593.587,E2 -26593.587} C_VEL
LIN {X 0,Y 129.83,Z 586.988,A -85,B 0,C 180,E1 -26598.099,E2 -26598.099} C_VEL
LIN {X 0,Y 136.584,Z 579.62,A -85,B 0,C 180,E1 -26601.521,E2 -26601.521} C_VEL
LIN {X 0,Y 142.864,Z 572.228,A -85,B 0,C 180,E1 -26604.26,E2 -26604.26} C_VEL
LIN {X 0,Y 150.667,Z 562.086,A -85,B 0,C 180,E1 -26607.098,E2 -26607.098} C_VEL
LIN {X 0,Y 158.703,Z 550.005,A -85,B 0,C 180,E1 -26609.713,E2 -26609.713} C_VEL
LIN {X 0,Y 165.665,Z 537.881,A -85,B 0,C 180,E1 -26611.672,E2 -26611.672} C_VEL
LIN {X 0,Y 171.919,Z 524.886,A -85,B 0,C 180,E1 -26613.333,E2 -26613.333} C_VEL
LIN {X 0,Y 177,Z 512.128,A -85,B 0,C 180,E1 -26614.594,E2 -26614.594} C_VEL
LIN {X 0,Y 181.737,Z 497.387,A -85,B 0,C 180,E1 -26615.667,E2 -26615.667} C_VEL
LIN {X 0,Y 185.287,Z 482.534,A -85,B 0,C 180,E1 -26616.454,E2 -26616.454} C_VEL
LIN {X 0,Y 187.73,Z 467.634,A -85,B 0,C 180,E1 -26616.96,E2 -26616.96} C_VEL
LIN {X 0,Y 191.592,Z 429.367,A -85,B 0,C 180,E1 -26617.931,E2 -26617.931} C_VEL
LIN {X 0,Y 189.162,Z 423.739,A -85,B 0,C 180,E1 -26620.465,E2 -26620.465} C_VEL
LIN {X 0,Y 186.575,Z 418.289,A -85,B 0,C 180,E1 -26623.589,E2 -26623.589} C_VEL
LIN {X 0,Y 184.682,Z 414.487,A -85,B 0,C 180,E1 -26626.356,E2 -26626.356} C_VEL
LIN {X 0,Y 183.658,Z 412.506,A -85,B 0,C 180,E1 -26628.13,E2 -26628.13} C_VEL
LIN {X 0,Y 182.194,Z 409.384,A -85,B 0,C 180,E1 -26631.403,E2 -26631.403} C_VEL
LIN {X 0,Y 180.845,Z 405.605,A -85,B 0,C 180,E1 -26637.494,E2 -26637.494} C_VEL
LIN {X 0,Y 180.77,Z 405.369,A -85,B 0,C 180,E1 -26641.114,E2 -26641.114} C_VEL
LIN {X 0,Y 180.857,Z 405.738,A -85,B 0,C 180,E1 -26642.366,E2 -26642.366} C_VEL
LIN {X 0,Y 182.495,Z 409.978,A -85,B 0,C 180,E1 -26649.001,E2 -26649.001} C_VEL
LIN {X 0,Y 184.466,Z 414.069,A -85,B 0,C 180,E1 -26652.934,E2 -26652.934} C_VEL
LIN {X 0,Y 186.604,Z 418.302,A -85,B 0,C 180,E1 -26656.086,E2 -26656.086} C_VEL
LIN {X 0,Y 188.866,Z 423.215,A -85,B 0,C 180,E1 -26658.861,E2 -26658.861} C_VEL
LIN {X 0,Y 191.235,Z 430.55,A -85,B 0,C 180,E1 -26661.562,E2 -26661.562} C_VEL
LIN {X 0,Y 191.47,Z 431.354,A -85,B 0,C 180,E1 -26661.816,E2 -26661.816} C_VEL
LIN {X 0,Y 186.802,Z 476.037,A -85,B 0,C 180,E1 -26662.929,E2 -26662.929} C_VEL
LIN {X 0,Y 183.902,Z 491.337,A -85,B 0,C 180,E1 -26663.486,E2 -26663.486} C_VEL
LIN {X 0,Y 179.768,Z 506.55,A -85,B 0,C 180,E1 -26664.304,E2 -26664.304} C_VEL
LIN {X 0,Y 174.914,Z 520.267,A -85,B 0,C 180,E1 -26665.308,E2 -26665.308} C_VEL
LIN {X 0,Y 169.046,Z 533.71,A -85,B 0,C 180,E1 -26666.642,E2 -26666.642} C_VEL
LIN {X 0,Y 162.285,Z 546.615,A -85,B 0,C 180,E1 -26668.329,E2 -26668.329} C_VEL
LIN {X 0,Y 154.238,Z 559.813,A -85,B 0,C 180,E1 -26670.68,E2 -26670.68} C_VEL
LIN {X 0,Y 145.434,Z 571.974,A -85,B 0,C 180,E1 -26673.533,E2 -26673.533} C_VEL
LIN {X 0,Y 136.527,Z 582.805,A -85,B 0,C 180,E1 -26677.072,E2 -26677.072} C_VEL
LIN {X 0,Y 128.201,Z 591.885,A -85,B 0,C 180,E1 -26681.135,E2 -26681.135} C_VEL
LIN {X 0,Y 120.825,Z 599.34,A -85,B 0,C 180,E1 -26685.735,E2 -26685.735} C_VEL
LIN {X 0,Y 113.168,Z 606.337,A -85,B 0,C 180,E1 -26691.61,E2 -26691.61} C_VEL
LIN {X 0,Y 106.99,Z 611.852,A -85,B 0,C 180,E1 -26698.298,E2 -26698.298} C_VEL
LIN {X 0,Y 102.351,Z 616.031,A -85,B 0,C 180,E1 -26705.671,E2 -26705.671} C_VEL
LIN {X 0,Y 99.324,Z 618.969,A -85,B 0,C 180,E1 -26713.559,E2 -26713.559} C_VEL
LIN {X 0,Y 98.013,Z 620.732,A -85,B 0,C 180,E1 -26721.755,E2 -26721.755} C_VEL
LIN {X 0,Y 98.071,Z 621.345,A -85,B 0,C 180,E1 -26730,E2 -26730} C_VEL
LIN {X 0,Y 98.006,Z 620.712,A -85,B 0,C 180,E1 -26738.246,E2 -26738.246} C_VEL
LIN {X 0,Y 99.296,Z 618.921,A -85,B 0,C 180,E1 -26746.446,E2 -26746.446} C_VEL
LIN {X 0,Y 100.01,Z 618.119,A -85,B 0,C 180,E1 -26748.872,E2 -26748.872} C_VEL
LIN {X 0,Y 100.585,Z 616.98,A -85,B 0,C 180,E1 -26752.164,E2 -26752.164} C_VEL
LIN {X 0,Y 100.416,Z 614.719,A -85,B 0,C 180,E1 -26757.67,E2 -26757.67} C_VEL
LIN {X 0,Y 100.744,Z 612.565,A -85,B 0,C 180,E1 -26762.031,E2 -26762.031} C_VEL
LIN {X 0,Y 102.077,Z 610.681,A -85,B 0,C 180,E1 -26765.112,E2 -26765.112} C_VEL
LIN {X 0,Y 102.823,Z 609.999,A -85,B 0,C 180,E1 -26766.06,E2 -26766.06} C_VEL
LIN {X 0,Y 109.568,Z 604.382,A -85,B 0,C 180,E1 -26772.336,E2 -26772.336} C_VEL
LIN {X 0,Y 117.975,Z 596.943,A -85,B 0,C 180,E1 -26778.127,E2 -26778.127} C_VEL
LIN {X 0,Y 126.046,Z 588.984,A -85,B 0,C 180,E1 -26782.61,E2 -26782.61} C_VEL
LIN {X 0,Y 134.945,Z 579.447,A -85,B 0,C 180,E1 -26786.435,E2 -26786.435} C_VEL
LIN {X 0,Y 142.964,Z 569.732,A -85,B 0,C 180,E1 -26789.346,E2 -26789.346} C_VEL
LIN {X 0,Y 151.414,Z 558.207,A -85,B 0,C 180,E1 -26791.869,E2 -26791.869} C_VEL
LIN {X 0,Y 158.582,Z 546.806,A -85,B 0,C 180,E1 -26793.819,E2 -26793.819} C_VEL
LIN {X 0,Y 165.206,Z 534.546,A -85,B 0,C 180,E1 -26795.406,E2 -26795.406} C_VEL
LIN {X 0,Y 171.238,Z 521.286,A -85,B 0,C 180,E1 -26796.678,E2 -26796.678} C_VEL
LIN {X 0,Y 176.585,Z 506.77,A -85,B 0,C 180,E1 -26797.715,E2 -26797.715} C_VEL
LIN {X 0,Y 180.811,Z 491.706,A -85,B 0,C 180,E1 -26798.498,E2 -26798.498} C_VEL
LIN {X 0,Y 183.867,Z 476.04,A -85,B 0,C 180,E1 -26799.059,E2 -26799.059} C_VEL
LIN {X 0,Y 188.336,Z 434.355,A -85,B 0,C 180,E1 -26800.092,E2 -26800.092} C_VEL
LIN {X 0,Y 186.424,Z 428.135,A -85,B 0,C 180,E1 -26802.518,E2 -26802.518} C_VEL
LIN {X 0,Y 183.986,Z 422.744,A -85,B 0,C 180,E1 -26805.886,E2 -26805.886} C_VEL
LIN {X 0,Y 182.118,Z 418.871,A -85,B 0,C 180,E1 -26809.157,E2 -26809.157} C_VEL
LIN {X 0,Y 180.86,Z 416.014,A -85,B 0,C 180,E1 -26812.183,E2 -26812.183} C_VEL
LIN {X 0,Y 179.63,Z 412.284,A -85,B 0,C 180,E1 -26818.406,E2 -26818.406} C_VEL
LIN {X 0,Y 179.671,Z 412.391,A -85,B 0,C 180,E1 -26822.522,E2 -26822.522} C_VEL
LIN {X 0,Y 180.895,Z 416.141,A -85,B 0,C 180,E1 -26828.378,E2 -26828.378} C_VEL
LIN {X 0,Y 182.966,Z 420.648,A -85,B 0,C 180,E1 -26832.89,E2 -26832.89} C_VEL
LIN {X 0,Y 185.007,Z 424.927,A -85,B 0,C 180,E1 -26836.058,E2 -26836.058} C_VEL
LIN {X 0,Y 187.895,Z 431.551,A -85,B 0,C 180,E1 -26839.672,E2 -26839.672} C_VEL
LIN {X 0,Y 188.416,Z 432.814,A -85,B 0,C 180,E1 -26840.254,E2 -26840.254} C_VEL
LIN {X 0,Y 184.327,Z 471.514,A -85,B 0,C 180,E1 -26841.235,E2 -26841.235} C_VEL
LIN {X 0,Y 181.45,Z 486.934,A -85,B 0,C 180,E1 -26841.823,E2 -26841.823} C_VEL
LIN {X 0,Y 177.501,Z 501.616,A -85,B 0,C 180,E1 -26842.63,E2 -26842.63} C_VEL
LIN {X 0,Y 172.657,Z 515.399,A -85,B 0,C 180,E1 -26843.675,E2 -26843.675} C_VEL
LIN {X 0,Y 166.148,Z 530.338,A -85,B 0,C 180,E1 -26845.232,E2 -26845.232} C_VEL
LIN {X 0,Y 159.622,Z 542.656,A -85,B 0,C 180,E1 -26846.93,E2 -26846.93} C_VEL
LIN {X 0,Y 151.799,Z 555.055,A -85,B 0,C 180,E1 -26849.091,E2 -26849.091} C_VEL
LIN {X 0,Y 144.27,Z 565.432,A -85,B 0,C 180,E1 -26851.518,E2 -26851.518} C_VEL
LIN {X 0,Y 136.285,Z 575.062,A -85,B 0,C 180,E1 -26854.404,E2 -26854.404} C_VEL
LIN {X 0,Y 127.71,Z 584.487,A -85,B 0,C 180,E1 -26858.356,E2 -26858.356} C_VEL
LIN {X 0,Y 119.522,Z 592.338,A -85,B 0,C 180,E1 -26862.694,E2 -26862.694} C_VEL
LIN {X 0,Y 111.144,Z 599.661,A -85,B 0,C 180,E1 -26868.4,E2 -26868.4} C_VEL
LIN {X 0,Y 104.029,Z 605.46,A -85,B 0,C 180,E1 -26874.955,E2 -26874.955} C_VEL
LIN {X 0,Y 99.64,Z 608.89,A -85,B 0,C 180,E1 -26880.415,E2 -26880.415} C_VEL
LIN {X 0,Y 95.121,Z 612.354,A -85,B 0,C 180,E1 -26888.321,E2 -26888.321} C_VEL
LIN {X 0,Y 92.315,Z 614.633,A -85,B 0,C 180,E1 -26896.798,E2 -26896.798} C_VEL
LIN {X 0,Y 91.106,Z 615.786,A -85,B 0,C 180,E1 -26905.576,E2 -26905.576} C_VEL
LIN {X 0,Y 91.056,Z 615.937,A -85,B 0,C 180,E1 -26910,E2 -26910} C_VEL
LIN {X 0,Y 91.541,Z 615.377,A -85,B 0,C 180,E1 -26918.832,E2 -26918.832} C_VEL
LIN {X 0,Y 93.474,Z 613.708,A -85,B 0,C 180,E1 -26927.502,E2 -26927.502} C_VEL
LIN {X 0,Y 97.066,Z 610.883,A -85,B 0,C 180,E1 -26935.748,E2 -26935.748} C_VEL
LIN {X 0,Y 102.429,Z 606.826,A -85,B 0,C 180,E1 -26943.291,E2 -26943.291} C_VEL
LIN {X 0,Y 109.221,Z 601.442,A -85,B 0,C 180,E1 -26950.049,E2 -26950.049} C_VEL
LIN {X 0,Y 117.258,Z 594.575,A -85,B 0,C 180,E1 -26955.99,E2 -26955.99} C_VEL
LIN {X 0,Y 125.203,Z 587.19,A -85,B 0,C 180,E1 -26960.516,E2 -26960.516} C_VEL
LIN {X 0,Y 132.878,Z 579.128,A -85,B 0,C 180,E1 -26964.243,E2 -26964.243} C_VEL
LIN {X 0,Y 141.474,Z 569.195,A -85,B 0,C 180,E1 -26967.617,E2 -26967.617} C_VEL
LIN {X 0,Y 149.665,Z 558.464,A -85,B 0,C 180,E1 -26970.308,E2 -26970.308} C_VEL
LIN {X 0,Y 157.385,Z 546.747,A -85,B 0,C 180,E1 -26972.559,E2 -26972.559} C_VEL
LIN {X 0,Y 164.541,Z 534.02,A -85,B 0,C 180,E1 -26974.422,E2 -26974.422} C_VEL
LIN {X 0,Y 170.409,Z 521.567,A -85,B 0,C 180,E1 -26975.846,E2 -26975.846} C_VEL
LIN {X 0,Y 175.565,Z 508.267,A -85,B 0,C 180,E1 -26977.026,E2 -26977.026} C_VEL
LIN {X 0,Y 180.038,Z 493.598,A -85,B 0,C 180,E1 -26977.985,E2 -26977.985} C_VEL
LIN {X 0,Y 183.504,Z 478.11,A -85,B 0,C 180,E1 -26978.665,E2 -26978.665} C_VEL
LIN {X 0,Y 185.725,Z 462.381,A -85,B 0,C 180,E1 -26979.112,E2 -26979.112} C_VEL
LIN {X 0,Y 188.672,Z 433.067,A -85,B 0,C 180,E1 -26979.848,E2 -26979.848} C_VEL
LIN {X 0,Y 185.663,Z 426.037,A -85,B 0,C 180,E1 -26983.507,E2 -26983.507} C_VEL
LIN {X 0,Y 183.443,Z 421.343,A -85,B 0,C 180,E1 -26986.851,E2 -26986.851} C_VEL
LIN {X 0,Y 182.351,Z 419.071,A -85,B 0,C 180,E1 -26988.889,E2 -26988.889} C_VEL
LIN {X 0,Y 181.138,Z 416.276,A -85,B 0,C 180,E1 -26991.844,E2 -26991.844} C_VEL
LIN {X 0,Y 179.919,Z 412.433,A -85,B 0,C 180,E1 -26998.321,E2 -26998.321} C_VEL
LIN {X 0,Y 179.95,Z 412.565,A -85,B 0,C 180,E1 -27001.818,E2 -27001.818} C_VEL
LIN {X 0,Y 181.445,Z 416.937,A -85,B 0,C 180,E1 -27008.632,E2 -27008.632} C_VEL
LIN {X 0,Y 183.177,Z 420.765,A -85,B 0,C 180,E1 -27012.322,E2 -27012.322} C_VEL
LIN {X 0,Y 184.854,Z 424.333,A -85,B 0,C 180,E1 -27015.011,E2 -27015.011} C_VEL
LIN {X 0,Y 186.98,Z 429.207,A -85,B 0,C 180,E1 -27017.852,E2 -27017.852} C_VEL
LIN {X 0,Y 188.558,Z 434.495,A -85,B 0,C 180,E1 -27019.855,E2 -27019.855} C_VEL
LIN {X 0,Y 184.258,Z 475.126,A -85,B 0,C 180,E1 -27020.863,E2 -27020.863} C_VEL
LIN {X 0,Y 181.19,Z 491.144,A -85,B 0,C 180,E1 -27021.426,E2 -27021.426} C_VEL
LIN {X 0,Y 176.964,Z 506.354,A -85,B 0,C 180,E1 -27022.209,E2 -27022.209} C_VEL
LIN {X 0,Y 171.991,Z 520.07,A -85,B 0,C 180,E1 -27023.164,E2 -27023.164} C_VEL
LIN {X 0,Y 165.985,Z 533.512,A -85,B 0,C 180,E1 -27024.451,E2 -27024.451} C_VEL
LIN {X 0,Y 159.306,Z 545.911,A -85,B 0,C 180,E1 -27025.993,E2 -27025.993} C_VEL
LIN {X 0,Y 151.443,Z 558.54,A -85,B 0,C 180,E1 -27028.151,E2 -27028.151} C_VEL
LIN {X 0,Y 142.981,Z 570.013,A -85,B 0,C 180,E1 -27030.665,E2 -27030.665} C_VEL
LIN {X 0,Y 134.942,Z 579.678,A -85,B 0,C 180,E1 -27033.562,E2 -27033.562} C_VEL
LIN {X 0,Y 126.04,Z 589.177,A -85,B 0,C 180,E1 -27037.386,E2 -27037.386} C_VEL
LIN {X 0,Y 117.941,Z 597.103,A -85,B 0,C 180,E1 -27041.854,E2 -27041.854} C_VEL
LIN {X 0,Y 109.539,Z 604.506,A -85,B 0,C 180,E1 -27047.65,E2 -27047.65} C_VEL
LIN {X 0,Y 102.476,Z 610.39,A -85,B 0,C 180,E1 -27054.343,E2 -27054.343} C_VEL
LIN {X 0,Y 98.206,Z 613.897,A -85,B 0,C 180,E1 -27059.938,E2 -27059.938} C_VEL
LIN {X 0,Y 93.938,Z 617.445,A -85,B 0,C 180,E1 -27068.033,E2 -27068.033} C_VEL
LIN {X 0,Y 91.52,Z 619.791,A -85,B 0,C 180,E1 -27076.681,E2 -27076.681} C_VEL
LIN {X 0,Y 90.809,Z 620.98,A -85,B 0,C 180,E1 -27085.561,E2 -27085.561} C_VEL
LIN {X 0,Y 90.969,Z 621.142,A -85,B 0,C 180,E1 -27090,E2 -27090} C_VEL
LIN {X 0,Y 90.951,Z 620.508,A -85,B 0,C 180,E1 -27098.89,E2 -27098.89} C_VEL
LIN {X 0,Y 92.442,Z 618.716,A -85,B 0,C 180,E1 -27107.704,E2 -27107.704} C_VEL
LIN {X 0,Y 95.787,Z 615.754,A -85,B 0,C 180,E1 -27116.117,E2 -27116.117} C_VEL
LIN {X 0,Y 100.899,Z 611.555,A -85,B 0,C 180,E1 -27123.864,E2 -27123.864} C_VEL
LIN {X 0,Y 102.823,Z 609.999,A -85,B 0,C 180,E1 -27126.06,E2 -27126.06} C_VEL
LIN {X 0,Y 104.858,Z 607.897,A -85,B 0,C 180,E1 -27128.886,E2 -27128.886} C_VEL
LIN {X 0,Y 107.184,Z 604.177,A -85,B 0,C 180,E1 -27133.686,E2 -27133.686} C_VEL
LIN {X 0,Y 110.017,Z 600.059,A -85,B 0,C 180,E1 -27138.202,E2 -27138.202} C_VEL
LIN {X 0,Y 112.734,Z 597.239,A -85,B 0,C 180,E1 -27140.491,E2 -27140.491} C_VEL
LIN {X 0,Y 121.823,Z 588.777,A -85,B 0,C 180,E1 -27145.292,E2 -27145.292} C_VEL
LIN {X 0,Y 131.12,Z 579.24,A -85,B 0,C 180,E1 -27149.045,E2 -27149.045} C_VEL
LIN {X 0,Y 139.465,Z 569.525,A -85,B 0,C 180,E1 -27151.866,E2 -27151.866} C_VEL
LIN {X 0,Y 148.18,Z 558,A -85,B 0,C 180,E1 -27154.306,E2 -27154.306} C_VEL
LIN {X 0,Y 156.309,Z 545.302,A -85,B 0,C 180,E1 -27156.36,E2 -27156.36} C_VEL
LIN {X 0,Y 163.144,Z 532.795,A -85,B 0,C 180,E1 -27157.844,E2 -27157.844} C_VEL
LIN {X 0,Y 169.331,Z 519.229,A -85,B 0,C 180,E1 -27159.039,E2 -27159.039} C_VEL
LIN {X 0,Y 174.411,Z 505.417,A -85,B 0,C 180,E1 -27159.945,E2 -27159.945} C_VEL
LIN {X 0,Y 178.718,Z 489.907,A -85,B 0,C 180,E1 -27160.693,E2 -27160.693} C_VEL
LIN {X 0,Y 181.624,Z 474.733,A -85,B 0,C 180,E1 -27161.19,E2 -27161.19} C_VEL
LIN {X 0,Y 185.646,Z 437.648,A -85,B 0,C 180,E1 -27162.089,E2 -27162.089} C_VEL
LIN {X 0,Y 184.416,Z 433.714,A -85,B 0,C 180,E1 -27163.819,E2 -27163.819} C_VEL
LIN {X 0,Y 182.312,Z 428.77,A -85,B 0,C 180,E1 -27167.052,E2 -27167.052} C_VEL
LIN {X 0,Y 180.776,Z 425.293,A -85,B 0,C 180,E1 -27170.066,E2 -27170.066} C_VEL
LIN {X 0,Y 179.812,Z 422.9,A -85,B 0,C 180,E1 -27172.632,E2 -27172.632} C_VEL
LIN {X 0,Y 178.761,Z 419.364,A -85,B 0,C 180,E1 -27178.398,E2 -27178.398} C_VEL
LIN {X 0,Y 178.782,Z 419.371,A -85,B 0,C 180,E1 -27182.253,E2 -27182.253} C_VEL
LIN {X 0,Y 179.821,Z 422.992,A -85,B 0,C 180,E1 -27187.862,E2 -27187.862} C_VEL
LIN {X 0,Y 181.613,Z 427.174,A -85,B 0,C 180,E1 -27192.121,E2 -27192.121} C_VEL
LIN {X 0,Y 183.619,Z 431.691,A -85,B 0,C 180,E1 -27195.47,E2 -27195.47} C_VEL
LIN {X 0,Y 185.697,Z 436.793,A -85,B 0,C 180,E1 -27198.301,E2 -27198.301} C_VEL
LIN {X 0,Y 181.775,Z 472.349,A -85,B 0,C 180,E1 -27199.171,E2 -27199.171} C_VEL
LIN {X 0,Y 178.933,Z 487.147,A -85,B 0,C 180,E1 -27199.712,E2 -27199.712} C_VEL
LIN {X 0,Y 174.901,Z 501.826,A -85,B 0,C 180,E1 -27200.49,E2 -27200.49} C_VEL
LIN {X 0,Y 169.931,Z 515.609,A -85,B 0,C 180,E1 -27201.483,E2 -27201.483} C_VEL
LIN {X 0,Y 163.531,Z 529.95,A -85,B 0,C 180,E1 -27202.901,E2 -27202.901} C_VEL
LIN {X 0,Y 156.533,Z 542.864,A -85,B 0,C 180,E1 -27204.611,E2 -27204.611} C_VEL
LIN {X 0,Y 148.48,Z 555.261,A -85,B 0,C 180,E1 -27206.699,E2 -27206.699} C_VEL
LIN {X 0,Y 140.68,Z 565.639,A -85,B 0,C 180,E1 -27209.046,E2 -27209.046} C_VEL
LIN {X 0,Y 132.393,Z 575.268,A -85,B 0,C 180,E1 -27211.862,E2 -27211.862} C_VEL
LIN {X 0,Y 125.928,Z 582.214,A -85,B 0,C 180,E1 -27214.597,E2 -27214.597} C_VEL
LIN {X 0,Y 117.156,Z 590.462,A -85,B 0,C 180,E1 -27218.756,E2 -27218.756} C_VEL
LIN {X 0,Y 108.036,Z 598.202,A -85,B 0,C 180,E1 -27224.311,E2 -27224.311} C_VEL
LIN {X 0,Y 100.069,Z 604.354,A -85,B 0,C 180,E1 -27230.798,E2 -27230.798} C_VEL
LIN {X 0,Y 93.501,Z 609.095,A -85,B 0,C 180,E1 -27238.255,E2 -27238.255} C_VEL
LIN {X 0,Y 88.528,Z 612.559,A -85,B 0,C 180,E1 -27246.614,E2 -27246.614} C_VEL
LIN {X 0,Y 85.411,Z 614.837,A -85,B 0,C 180,E1 -27255.709,E2 -27255.709} C_VEL
LIN {X 0,Y 84.05,Z 615.989,A -85,B 0,C 180,E1 -27265.204,E2 -27265.204} C_VEL
LIN {X 0,Y 83.956,Z 616.14,A -85,B 0,C 180,E1 -27270,E2 -27270} C_VEL
LIN {X 0,Y 84.514,Z 615.581,A -85,B 0,C 180,E1 -27279.573,E2 -27279.573} C_VEL
LIN {X 0,Y 86.703,Z 613.911,A -85,B 0,C 180,E1 -27288.919,E2 -27288.919} C_VEL
LIN {X 0,Y 90.693,Z 611.086,A -85,B 0,C 180,E1 -27297.706,E2 -27297.706} C_VEL
LIN {X 0,Y 96.539,Z 607.029,A -85,B 0,C 180,E1 -27305.618,E2 -27305.618} C_VEL
LIN {X 0,Y 103.86,Z 601.644,A -85,B 0,C 180,E1 -27312.583,E2 -27312.583} C_VEL
LIN {X 0,Y 112.411,Z 594.777,A -85,B 0,C 180,E1 -27318.61,E2 -27318.61} C_VEL
LIN {X 0,Y 120.812,Z 587.391,A -85,B 0,C 180,E1 -27323.116,E2 -27323.116} C_VEL
LIN {X 0,Y 129.396,Z 578.709,A -85,B 0,C 180,E1 -27327.102,E2 -27327.102} C_VEL
LIN {X 0,Y 137.801,Z 569.395,A -85,B 0,C 180,E1 -27330.111,E2 -27330.111} C_VEL
LIN {X 0,Y 146.279,Z 558.664,A -85,B 0,C 180,E1 -27332.724,E2 -27332.724} C_VEL
LIN {X 0,Y 154.243,Z 546.947,A -85,B 0,C 180,E1 -27334.9,E2 -27334.9} C_VEL
LIN {X 0,Y 161.989,Z 533.489,A -85,B 0,C 180,E1 -27336.779,E2 -27336.779} C_VEL
LIN {X 0,Y 168.373,Z 520.004,A -85,B 0,C 180,E1 -27338.234,E2 -27338.234} C_VEL
LIN {X 0,Y 174.056,Z 505.081,A -85,B 0,C 180,E1 -27339.429,E2 -27339.429} C_VEL
LIN {X 0,Y 178.477,Z 489.987,A -85,B 0,C 180,E1 -27340.279,E2 -27340.279} C_VEL
LIN {X 0,Y 181.689,Z 474.405,A -85,B 0,C 180,E1 -27340.893,E2 -27340.893} C_VEL
LIN {X 0,Y 184.145,Z 454.413,A -85,B 0,C 180,E1 -27341.394,E2 -27341.394} C_VEL
LIN {X 0,Y 185.931,Z 437.015,A -85,B 0,C 180,E1 -27341.829,E2 -27341.829} C_VEL
LIN {X 0,Y 183.641,Z 431.41,A -85,B 0,C 180,E1 -27344.995,E2 -27344.995} C_VEL
LIN {X 0,Y 181.47,Z 426.387,A -85,B 0,C 180,E1 -27348.834,E2 -27348.834} C_VEL
LIN {X 0,Y 180.043,Z 423.102,A -85,B 0,C 180,E1 -27352.429,E2 -27352.429} C_VEL
LIN {X 0,Y 179.056,Z 419.459,A -85,B 0,C 180,E1 -27358.313,E2 -27358.313} C_VEL
LIN {X 0,Y 179.056,Z 419.616,A -85,B 0,C 180,E1 -27361.546,E2 -27361.546} C_VEL
LIN {X 0,Y 180.349,Z 423.812,A -85,B 0,C 180,E1 -27368.121,E2 -27368.121} C_VEL
LIN {X 0,Y 181.961,Z 427.594,A -85,B 0,C 180,E1 -27371.805,E2 -27371.805} C_VEL
LIN {X 0,Y 183.846,Z 431.864,A -85,B 0,C 180,E1 -27374.953,E2 -27374.953} C_VEL
LIN {X 0,Y 185.148,Z 435.248,A -85,B 0,C 180,E1 -27376.824,E2 -27376.824} C_VEL
LIN {X 0,Y 185.901,Z 437.932,A -85,B 0,C 180,E1 -27377.898,E2 -27377.898} C_VEL
LIN {X 0,Y 181.849,Z 474.939,A -85,B 0,C 180,E1 -27378.771,E2 -27378.771} C_VEL
LIN {X 0,Y 178.719,Z 490.95,A -85,B 0,C 180,E1 -27379.308,E2 -27379.308} C_VEL
LIN {X 0,Y 174.407,Z 506.158,A -85,B 0,C 180,E1 -27380.051,E2 -27380.051} C_VEL
LIN {X 0,Y 169.317,Z 519.872,A -85,B 0,C 180,E1 -27380.948,E2 -27380.948} C_VEL
LIN {X 0,Y 163.171,Z 533.314,A -85,B 0,C 180,E1 -27382.179,E2 -27382.179} C_VEL
LIN {X 0,Y 156.308,Z 545.71,A -85,B 0,C 180,E1 -27383.64,E2 -27383.64} C_VEL
LIN {X 0,Y 148.209,Z 558.34,A -85,B 0,C 180,E1 -27385.718,E2 -27385.718} C_VEL
LIN {X 0,Y 139.481,Z 569.812,A -85,B 0,C 180,E1 -27388.147,E2 -27388.147} C_VEL
LIN {X 0,Y 131.116,Z 579.476,A -85,B 0,C 180,E1 -27390.952,E2 -27390.952} C_VEL
LIN {X 0,Y 121.822,Z 588.974,A -85,B 0,C 180,E1 -27394.707,E2 -27394.707} C_VEL
LIN {X 0,Y 113.265,Z 596.899,A -85,B 0,C 180,E1 -27399.141,E2 -27399.141} C_VEL
LIN {X 0,Y 106.492,Z 602.629,A -85,B 0,C 180,E1 -27403.453,E2 -27403.453} C_VEL
LIN {X 0,Y 98.499,Z 608.861,A -85,B 0,C 180,E1 -27410.048,E2 -27410.048} C_VEL
LIN {X 0,Y 92.049,Z 613.692,A -85,B 0,C 180,E1 -27417.694,E2 -27417.694} C_VEL
LIN {X 0,Y 87.326,Z 617.241,A -85,B 0,C 180,E1 -27426.272,E2 -27426.272} C_VEL
LIN {X 0,Y 84.575,Z 619.587,A -85,B 0,C 180,E1 -27435.565,E2 -27435.565} C_VEL
LIN {X 0,Y 83.73,Z 620.777,A -85,B 0,C 180,E1 -27445.185,E2 -27445.185} C_VEL
LIN {X 0,Y 83.875,Z 620.939,A -85,B 0,C 180,E1 -27450,E2 -27450} C_VEL
LIN {X 0,Y 83.728,Z 620.77,A -85,B 0,C 180,E1 -27454.815,E2 -27454.815} C_VEL
LIN {X 0,Y 84.557,Z 619.552,A -85,B 0,C 180,E1 -27464.438,E2 -27464.438} C_VEL
LIN {X 0,Y 87.293,Z 617.179,A -85,B 0,C 180,E1 -27473.737,E2 -27473.737} C_VEL
LIN {X 0,Y 91.943,Z 613.607,A -85,B 0,C 180,E1 -27482.348,E2 -27482.348} C_VEL
LIN {X 0,Y 98.502,Z 608.754,A -85,B 0,C 180,E1 -27489.95,E2 -27489.95} C_VEL
LIN {X 0,Y 106.507,Z 602.484,A -85,B 0,C 180,E1 -27496.538,E2 -27496.538} C_VEL
LIN {X 0,Y 112.734,Z 597.239,A -85,B 0,C 180,E1 -27500.491,E2 -27500.491} C_VEL
LIN {X 0,Y 115.554,Z 594.32,A -85,B 0,C 180,E1 -27502.651,E2 -27502.651} C_VEL
LIN {X 0,Y 119.225,Z 589.342,A -85,B 0,C 180,E1 -27506.446,E2 -27506.446} C_VEL
LIN {X 0,Y 123.226,Z 583.914,A -85,B 0,C 180,E1 -27509.86,E2 -27509.86} C_VEL
LIN {X 0,Y 126.418,Z 580.271,A -85,B 0,C 180,E1 -27511.395,E2 -27511.395} C_VEL
LIN {X 0,Y 134.773,Z 571.096,A -85,B 0,C 180,E1 -27514.094,E2 -27514.094} C_VEL
LIN {X 0,Y 144.478,Z 558.865,A -85,B 0,C 180,E1 -27516.654,E2 -27516.654} C_VEL
LIN {X 0,Y 152.817,Z 546.389,A -85,B 0,C 180,E1 -27518.632,E2 -27518.632} C_VEL
LIN {X 0,Y 159.819,Z 534.131,A -85,B 0,C 180,E1 -27520.041,E2 -27520.041} C_VEL
LIN {X 0,Y 166.118,Z 520.868,A -85,B 0,C 180,E1 -27521.191,E2 -27521.191} C_VEL
LIN {X 0,Y 171.708,Z 506.35,A -85,B 0,C 180,E1 -27522.1,E2 -27522.1} C_VEL
LIN {X 0,Y 175.907,Z 492.045,A -85,B 0,C 180,E1 -27522.765,E2 -27522.765} C_VEL
LIN {X 0,Y 178.947,Z 477.546,A -85,B 0,C 180,E1 -27523.245,E2 -27523.245} C_VEL
LIN {X 0,Y 181.718,Z 455.194,A -85,B 0,C 180,E1 -27523.764,E2 -27523.764} C_VEL
LIN {X 0,Y 183.187,Z 441.294,A -85,B 0,C 180,E1 -27524.096,E2 -27524.096} C_VEL
LIN {X 0,Y 181.962,Z 437.786,A -85,B 0,C 180,E1 -27526.031,E2 -27526.031} C_VEL
LIN {X 0,Y 180.074,Z 433.07,A -85,B 0,C 180,E1 -27529.601,E2 -27529.601} C_VEL
LIN {X 0,Y 178.734,Z 429.688,A -85,B 0,C 180,E1 -27533.226,E2 -27533.226} C_VEL
LIN {X 0,Y 177.892,Z 426.448,A -85,B 0,C 180,E1 -27538.391,E2 -27538.391} C_VEL
LIN {X 0,Y 177.89,Z 426.402,A -85,B 0,C 180,E1 -27541.981,E2 -27541.981} C_VEL
LIN {X 0,Y 178.763,Z 429.828,A -85,B 0,C 180,E1 -27547.341,E2 -27547.341} C_VEL
LIN {X 0,Y 180.373,Z 433.914,A -85,B 0,C 180,E1 -27551.512,E2 -27551.512} C_VEL
LIN {X 0,Y 182.183,Z 438.329,A -85,B 0,C 180,E1 -27554.772,E2 -27554.772} C_VEL
LIN {X 0,Y 183.17,Z 440.912,A -85,B 0,C 180,E1 -27556.28,E2 -27556.28} C_VEL
LIN {X 0,Y 179.547,Z 472.742,A -85,B 0,C 180,E1 -27557.045,E2 -27557.045} C_VEL
LIN {X 0,Y 176.669,Z 487.36,A -85,B 0,C 180,E1 -27557.549,E2 -27557.549} C_VEL
LIN {X 0,Y 172.552,Z 502.036,A -85,B 0,C 180,E1 -27558.29,E2 -27558.29} C_VEL
LIN {X 0,Y 167.463,Z 515.818,A -85,B 0,C 180,E1 -27559.223,E2 -27559.223} C_VEL
LIN {X 0,Y 161.39,Z 529.129,A -85,B 0,C 180,E1 -27560.454,E2 -27560.454} C_VEL
LIN {X 0,Y 154.465,Z 541.784,A -85,B 0,C 180,E1 -27562.026,E2 -27562.026} C_VEL
LIN {X 0,Y 146.915,Z 553.34,A -85,B 0,C 180,E1 -27563.815,E2 -27563.815} C_VEL
LIN {X 0,Y 138.848,Z 564.07,A -85,B 0,C 180,E1 -27566.05,E2 -27566.05} C_VEL
LIN {X 0,Y 130.174,Z 573.997,A -85,B 0,C 180,E1 -27568.681,E2 -27568.681} C_VEL
LIN {X 0,Y 123.324,Z 581.078,A -85,B 0,C 180,E1 -27571.263,E2 -27571.263} C_VEL
LIN {X 0,Y 115.396,Z 588.452,A -85,B 0,C 180,E1 -27574.697,E2 -27574.697} C_VEL
LIN {X 0,Y 107.899,Z 594.749,A -85,B 0,C 180,E1 -27578.593,E2 -27578.593} C_VEL
LIN {X 0,Y 98.74,Z 601.67,A -85,B 0,C 180,E1 -27584.622,E2 -27584.622} C_VEL
LIN {X 0,Y 90.858,Z 607.098,A -85,B 0,C 180,E1 -27591.772,E2 -27591.772} C_VEL
LIN {X 0,Y 84.485,Z 611.186,A -85,B 0,C 180,E1 -27600.059,E2 -27600.059} C_VEL
LIN {X 0,Y 80.053,Z 614.045,A -85,B 0,C 180,E1 -27609.442,E2 -27609.442} C_VEL
LIN {X 0,Y 77.513,Z 615.755,A -85,B 0,C 180,E1 -27619.553,E2 -27619.553} C_VEL
LIN {X 0,Y 76.883,Z 616.343,A -85,B 0,C 180,E1 -27630,E2 -27630} C_VEL
LIN {X 0,Y 77.511,Z 615.784,A -85,B 0,C 180,E1 -27640.448,E2 -27640.448} C_VEL
LIN {X 0,Y 80.002,Z 614.114,A -85,B 0,C 180,E1 -27650.572,E2 -27650.572} C_VEL
LIN {X 0,Y 84.446,Z 611.289,A -85,B 0,C 180,E1 -27659.956,E2 -27659.956} C_VEL
LIN {X 0,Y 90.835,Z 607.232,A -85,B 0,C 180,E1 -27668.239,E2 -27668.239} C_VEL
LIN {X 0,Y 98.717,Z 601.847,A -85,B 0,C 180,E1 -27675.391,E2 -27675.391} C_VEL
LIN {X 0,Y 107.829,Z 594.98,A -85,B 0,C 180,E1 -27681.454,E2 -27681.454} C_VEL
LIN {X 0,Y 116.687,Z 587.592,A -85,B 0,C 180,E1 -27685.908,E2 -27685.908} C_VEL
LIN {X 0,Y 126.125,Z 578.49,A -85,B 0,C 180,E1 -27689.968,E2 -27689.968} C_VEL
LIN {X 0,Y 135.858,Z 567.976,A -85,B 0,C 180,E1 -27693.167,E2 -27693.167} C_VEL
LIN {X 0,Y 145.361,Z 555.927,A -85,B 0,C 180,E1 -27695.86,E2 -27695.86} C_VEL
LIN {X 0,Y 153.655,Z 543.617,A -85,B 0,C 180,E1 -27697.848,E2 -27697.848} C_VEL
LIN {X 0,Y 161.143,Z 530.253,A -85,B 0,C 180,E1 -27699.533,E2 -27699.533} C_VEL
LIN {X 0,Y 167.411,Z 516.666,A -85,B 0,C 180,E1 -27700.827,E2 -27700.827} C_VEL
LIN {X 0,Y 172.883,Z 501.858,A -85,B 0,C 180,E1 -27701.843,E2 -27701.843} C_VEL
LIN {X 0,Y 177.197,Z 486.219,A -85,B 0,C 180,E1 -27702.626,E2 -27702.626} C_VEL
LIN {X 0,Y 180.074,Z 471.199,A -85,B 0,C 180,E1 -27703.119,E2 -27703.119} C_VEL
LIN {X 0,Y 183.399,Z 441.105,A -85,B 0,C 180,E1 -27703.869,E2 -27703.869} C_VEL
LIN {X 0,Y 181.406,Z 435.928,A -85,B 0,C 180,E1 -27707.128,E2 -27707.128} C_VEL
LIN {X 0,Y 179.89,Z 432.345,A -85,B 0,C 180,E1 -27710.3,E2 -27710.3} C_VEL
LIN {X 0,Y 178.991,Z 429.95,A -85,B 0,C 180,E1 -27712.952,E2 -27712.952} C_VEL
LIN {X 0,Y 178.157,Z 426.478,A -85,B 0,C 180,E1 -27718.87,E2 -27718.87} C_VEL
LIN {X 0,Y 178.168,Z 426.747,A -85,B 0,C 180,E1 -27721.412,E2 -27721.412} C_VEL
LIN {X 0,Y 179.281,Z 430.685,A -85,B 0,C 180,E1 -27727.636,E2 -27727.636} C_VEL
LIN {X 0,Y 180.723,Z 434.373,A -85,B 0,C 180,E1 -27731.212,E2 -27731.212} C_VEL
LIN {X 0,Y 182.354,Z 438.311,A -85,B 0,C 180,E1 -27734.152,E2 -27734.152} C_VEL
LIN {X 0,Y 183.446,Z 441.515,A -85,B 0,C 180,E1 -27735.881,E2 -27735.881} C_VEL
LIN {X 0,Y 179.619,Z 475.186,A -85,B 0,C 180,E1 -27736.64,E2 -27736.64} C_VEL
LIN {X 0,Y 176.5,Z 490.757,A -85,B 0,C 180,E1 -27737.133,E2 -27737.133} C_VEL
LIN {X 0,Y 172.103,Z 505.962,A -85,B 0,C 180,E1 -27737.831,E2 -27737.831} C_VEL
LIN {X 0,Y 166.912,Z 519.675,A -85,B 0,C 180,E1 -27738.673,E2 -27738.673} C_VEL
LIN {X 0,Y 160.618,Z 533.115,A -85,B 0,C 180,E1 -27739.826,E2 -27739.826} C_VEL
LIN {X 0,Y 153.593,Z 545.511,A -85,B 0,C 180,E1 -27741.207,E2 -27741.207} C_VEL
LIN {X 0,Y 145.255,Z 558.139,A -85,B 0,C 180,E1 -27743.18,E2 -27743.18} C_VEL
LIN {X 0,Y 136.267,Z 569.611,A -85,B 0,C 180,E1 -27745.506,E2 -27745.506} C_VEL
LIN {X 0,Y 127.588,Z 579.273,A -85,B 0,C 180,E1 -27748.199,E2 -27748.199} C_VEL
LIN {X 0,Y 117.892,Z 588.771,A -85,B 0,C 180,E1 -27751.845,E2 -27751.845} C_VEL
LIN {X 0,Y 108.885,Z 596.696,A -85,B 0,C 180,E1 -27756.216,E2 -27756.216} C_VEL
LIN {X 0,Y 101.709,Z 602.426,A -85,B 0,C 180,E1 -27760.53,E2 -27760.53} C_VEL
LIN {X 0,Y 93.103,Z 608.657,A -85,B 0,C 180,E1 -27767.207,E2 -27767.207} C_VEL
LIN {X 0,Y 86.065,Z 613.488,A -85,B 0,C 180,E1 -27775.138,E2 -27775.138} C_VEL
LIN {X 0,Y 80.815,Z 617.036,A -85,B 0,C 180,E1 -27784.227,E2 -27784.227} C_VEL
LIN {X 0,Y 77.655,Z 619.382,A -85,B 0,C 180,E1 -27794.246,E2 -27794.246} C_VEL
LIN {X 0,Y 76.624,Z 620.573,A -85,B 0,C 180,E1 -27804.737,E2 -27804.737} C_VEL
LIN {X 0,Y 76.771,Z 620.736,A -85,B 0,C 180,E1 -27810,E2 -27810} C_VEL
LIN {X 0,Y 76.88,Z 620.099,A -85,B 0,C 180,E1 -27820.534,E2 -27820.534} C_VEL
LIN {X 0,Y 78.905,Z 618.305,A -85,B 0,C 180,E1 -27830.871,E2 -27830.871} C_VEL
LIN {X 0,Y 83.127,Z 615.342,A -85,B 0,C 180,E1 -27840.481,E2 -27840.481} C_VEL
LIN {X 0,Y 89.343,Z 611.143,A -85,B 0,C 180,E1 -27848.998,E2 -27848.998} C_VEL
LIN {X 0,Y 97.25,Z 605.599,A -85,B 0,C 180,E1 -27856.274,E2 -27856.274} C_VEL
LIN {X 0,Y 106.507,Z 598.563,A -85,B 0,C 180,E1 -27862.355,E2 -27862.355} C_VEL
LIN {X 0,Y 116.557,Z 589.808,A -85,B 0,C 180,E1 -27867.579,E2 -27867.579} C_VEL
LIN {X 0,Y 126.418,Z 580.271,A -85,B 0,C 180,E1 -27871.395,E2 -27871.395} C_VEL
LIN {X 0,Y 129.647,Z 576.558,A -85,B 0,C 180,E1 -27872.821,E2 -27872.821} C_VEL
LIN {X 0,Y 137.374,Z 565.01,A -85,B 0,C 180,E1 -27877.652,E2 -27877.652} C_VEL
LIN {X 0,Y 140.254,Z 560.787,A -85,B 0,C 180,E1 -27878.88,E2 -27878.88} C_VEL
LIN {X 0,Y 141.316,Z 559.31,A -85,B 0,C 180,E1 -27879.189,E2 -27879.189} C_VEL
LIN {X 0,Y 149.585,Z 547.419,A -85,B 0,C 180,E1 -27880.999,E2 -27880.999} C_VEL
LIN {X 0,Y 157.531,Z 533.923,A -85,B 0,C 180,E1 -27882.475,E2 -27882.475} C_VEL
LIN {X 0,Y 163.962,Z 520.659,A -85,B 0,C 180,E1 -27883.545,E2 -27883.545} C_VEL
LIN {X 0,Y 169.659,Z 506.14,A -85,B 0,C 180,E1 -27884.384,E2 -27884.384} C_VEL
LIN {X 0,Y 174.13,Z 491.068,A -85,B 0,C 180,E1 -27885.039,E2 -27885.039} C_VEL
LIN {X 0,Y 177.328,Z 475.627,A -85,B 0,C 180,E1 -27885.496,E2 -27885.496} C_VEL
LIN {X 0,Y 180.893,Z 445.391,A -85,B 0,C 180,E1 -27886.165,E2 -27886.165} C_VEL
LIN {X 0,Y 179.406,Z 441.362,A -85,B 0,C 180,E1 -27888.991,E2 -27888.991} C_VEL
LIN {X 0,Y 178.377,Z 438.549,A -85,B 0,C 180,E1 -27891.504,E2 -27891.504} C_VEL
LIN {X 0,Y 177.688,Z 436.574,A -85,B 0,C 180,E1 -27893.756,E2 -27893.756} C_VEL
LIN {X 0,Y 176.979,Z 433.374,A -85,B 0,C 180,E1 -27899.191,E2 -27899.191} C_VEL
LIN {X 0,Y 177.004,Z 433.623,A -85,B 0,C 180,E1 -27901.991,E2 -27901.991} C_VEL
LIN {X 0,Y 177.958,Z 437.355,A -85,B 0,C 180,E1 -27907.66,E2 -27907.66} C_VEL
LIN {X 0,Y 179.209,Z 440.822,A -85,B 0,C 180,E1 -27911.022,E2 -27911.022} C_VEL
LIN {X 0,Y 180.661,Z 444.61,A -85,B 0,C 180,E1 -27913.857,E2 -27913.857} C_VEL
LIN {X 0,Y 180.871,Z 445.296,A -85,B 0,C 180,E1 -27914.24,E2 -27914.24} C_VEL
LIN {X 0,Y 177.578,Z 473.092,A -85,B 0,C 180,E1 -27914.866,E2 -27914.866} C_VEL
LIN {X 0,Y 174.663,Z 487.573,A -85,B 0,C 180,E1 -27915.331,E2 -27915.331} C_VEL
LIN {X 0,Y 170.461,Z 502.246,A -85,B 0,C 180,E1 -27916.027,E2 -27916.027} C_VEL
LIN {X 0,Y 165.261,Z 516.027,A -85,B 0,C 180,E1 -27916.898,E2 -27916.898} C_VEL
LIN {X 0,Y 158.806,Z 529.819,A -85,B 0,C 180,E1 -27918.101,E2 -27918.101} C_VEL
LIN {X 0,Y 151.17,Z 543.278,A -85,B 0,C 180,E1 -27919.71,E2 -27919.71} C_VEL
LIN {X 0,Y 142.656,Z 555.675,A -85,B 0,C 180,E1 -27921.588,E2 -27921.588} C_VEL
LIN {X 0,Y 134.367,Z 566.05,A -85,B 0,C 180,E1 -27923.751,E2 -27923.751} C_VEL
LIN {X 0,Y 125.46,Z 575.68,A -85,B 0,C 180,E1 -27926.33,E2 -27926.33} C_VEL
LIN {X 0,Y 118.389,Z 582.628,A -85,B 0,C 180,E1 -27928.885,E2 -27928.885} C_VEL
LIN {X 0,Y 108.793,Z 590.874,A -85,B 0,C 180,E1 -27932.884,E2 -27932.884} C_VEL
LIN {X 0,Y 98.602,Z 598.613,A -85,B 0,C 180,E1 -27938.37,E2 -27938.37} C_VEL
LIN {X 0,Y 89.451,Z 604.765,A -85,B 0,C 180,E1 -27945.001,E2 -27945.001} C_VEL
LIN {X 0,Y 81.721,Z 609.504,A -85,B 0,C 180,E1 -27952.988,E2 -27952.988} C_VEL
LIN {X 0,Y 75.636,Z 612.968,A -85,B 0,C 180,E1 -27962.317,E2 -27962.317} C_VEL
LIN {X 0,Y 71.703,Z 615.244,A -85,B 0,C 180,E1 -27972.9,E2 -27972.9} C_VEL
LIN {X 0,Y 69.918,Z 616.394,A -85,B 0,C 180,E1 -27984.231,E2 -27984.231} C_VEL
LIN {X 0,Y 69.783,Z 616.546,A -85,B 0,C 180,E1 -27990,E2 -27990} C_VEL
LIN {X 0,Y 70.543,Z 615.987,A -85,B 0,C 180,E1 -28001.493,E2 -28001.493} C_VEL
LIN {X 0,Y 73.369,Z 614.317,A -85,B 0,C 180,E1 -28012.529,E2 -28012.529} C_VEL
LIN {X 0,Y 78.356,Z 611.492,A -85,B 0,C 180,E1 -28022.558,E2 -28022.558} C_VEL
LIN {X 0,Y 85.35,Z 607.435,A -85,B 0,C 180,E1 -28031.203,E2 -28031.203} C_VEL
LIN {X 0,Y 93.83,Z 602.051,A -85,B 0,C 180,E1 -28038.503,E2 -28038.503} C_VEL
LIN {X 0,Y 103.544,Z 595.182,A -85,B 0,C 180,E1 -28044.535,E2 -28044.535} C_VEL
LIN {X 0,Y 112.855,Z 587.794,A -85,B 0,C 180,E1 -28048.898,E2 -28048.898} C_VEL
LIN {X 0,Y 122.42,Z 578.968,A -85,B 0,C 180,E1 -28052.748,E2 -28052.748} C_VEL
LIN {X 0,Y 131.299,Z 569.796,A -85,B 0,C 180,E1 -28055.496,E2 -28055.496} C_VEL
LIN {X 0,Y 140.335,Z 559.064,A -85,B 0,C 180,E1 -28057.889,E2 -28057.889} C_VEL
LIN {X 0,Y 148.776,Z 547.345,A -85,B 0,C 180,E1 -28059.859,E2 -28059.859} C_VEL
LIN {X 0,Y 156.581,Z 534.515,A -85,B 0,C 180,E1 -28061.486,E2 -28061.486} C_VEL
LIN {X 0,Y 162.85,Z 522.159,A -85,B 0,C 180,E1 -28062.709,E2 -28062.709} C_VEL
LIN {X 0,Y 168.404,Z 508.853,A -85,B 0,C 180,E1 -28063.705,E2 -28063.705} C_VEL
LIN {X 0,Y 173.2,Z 494.176,A -85,B 0,C 180,E1 -28064.512,E2 -28064.512} C_VEL
LIN {X 0,Y 176.777,Z 479.262,A -85,B 0,C 180,E1 -28065.076,E2 -28065.076} C_VEL
LIN {X 0,Y 179.204,Z 463.293,A -85,B 0,C 180,E1 -28065.471,E2 -28065.471} C_VEL
LIN {X 0,Y 181.119,Z 445.441,A -85,B 0,C 180,E1 -28065.907,E2 -28065.907} C_VEL
LIN {X 0,Y 179.588,Z 441.317,A -85,B 0,C 180,E1 -28068.859,E2 -28068.859} C_VEL
LIN {X 0,Y 178.264,Z 437.725,A -85,B 0,C 180,E1 -28072.353,E2 -28072.353} C_VEL
LIN {X 0,Y 177.738,Z 436.38,A -85,B 0,C 180,E1 -28074.312,E2 -28074.312} C_VEL
LIN {X 0,Y 177.294,Z 433.511,A -85,B 0,C 180,E1 -28078.864,E2 -28078.864} C_VEL
LIN {X 0,Y 177.287,Z 433.744,A -85,B 0,C 180,E1 -28081.135,E2 -28081.135} C_VEL
LIN {X 0,Y 178.209,Z 437.48,A -85,B 0,C 180,E1 -28087.079,E2 -28087.079} C_VEL
LIN {X 0,Y 179.558,Z 441.22,A -85,B 0,C 180,E1 -28090.714,E2 -28090.714} C_VEL
LIN {X 0,Y 181.159,Z 445.566,A -85,B 0,C 180,E1 -28093.806,E2 -28093.806} C_VEL
LIN {X 0,Y 177.717,Z 474.997,A -85,B 0,C 180,E1 -28094.448,E2 -28094.448} C_VEL
LIN {X 0,Y 174.541,Z 490.564,A -85,B 0,C 180,E1 -28094.907,E2 -28094.907} C_VEL
LIN {X 0,Y 170.066,Z 505.767,A -85,B 0,C 180,E1 -28095.557,E2 -28095.557} C_VEL
LIN {X 0,Y 164.774,Z 519.478,A -85,B 0,C 180,E1 -28096.331,E2 -28096.331} C_VEL
LIN {X 0,Y 158.351,Z 532.917,A -85,B 0,C 180,E1 -28097.409,E2 -28097.409} C_VEL
LIN {X 0,Y 151.158,Z 545.311,A -85,B 0,C 180,E1 -28098.684,E2 -28098.684} C_VEL
LIN {X 0,Y 142.594,Z 557.938,A -85,B 0,C 180,E1 -28100.541,E2 -28100.541} C_VEL
LIN {X 0,Y 133.358,Z 569.411,A -85,B 0,C 180,E1 -28102.746,E2 -28102.746} C_VEL
LIN {X 0,Y 124.377,Z 579.072,A -85,B 0,C 180,E1 -28105.303,E2 -28105.303} C_VEL
LIN {X 0,Y 114.285,Z 588.569,A -85,B 0,C 180,E1 -28108.802,E2 -28108.802} C_VEL
LIN {X 0,Y 104.814,Z 596.493,A -85,B 0,C 180,E1 -28113.057,E2 -28113.057} C_VEL
LIN {X 0,Y 94.765,Z 603.895,A -85,B 0,C 180,E1 -28118.86,E2 -28118.86} C_VEL
LIN {X 0,Y 85.896,Z 609.777,A -85,B 0,C 180,E1 -28125.937,E2 -28125.937} C_VEL
LIN {X 0,Y 80.27,Z 613.283,A -85,B 0,C 180,E1 -28132.203,E2 -28132.203} C_VEL
LIN {X 0,Y 74.43,Z 616.832,A -85,B 0,C 180,E1 -28141.829,E2 -28141.829} C_VEL
LIN {X 0,Y 70.793,Z 619.178,A -85,B 0,C 180,E1 -28152.673,E2 -28152.673} C_VEL
LIN {X 0,Y 69.537,Z 620.37,A -85,B 0,C 180,E1 -28164.199,E2 -28164.199} C_VEL
LIN {X 0,Y 69.666,Z 620.533,A -85,B 0,C 180,E1 -28170,E2 -28170} C_VEL
LIN {X 0,Y 69.861,Z 619.894,A -85,B 0,C 180,E1 -28181.607,E2 -28181.607} C_VEL
LIN {X 0,Y 72.251,Z 618.1,A -85,B 0,C 180,E1 -28192.897,E2 -28192.897} C_VEL
LIN {X 0,Y 77.027,Z 615.136,A -85,B 0,C 180,E1 -28203.191,E2 -28203.191} C_VEL
LIN {X 0,Y 83.884,Z 610.937,A -85,B 0,C 180,E1 -28212.085,E2 -28212.085} C_VEL
LIN {X 0,Y 92.429,Z 605.393,A -85,B 0,C 180,E1 -28219.495,E2 -28219.495} C_VEL
LIN {X 0,Y 102.26,Z 598.355,A -85,B 0,C 180,E1 -28225.558,E2 -28225.558} C_VEL
LIN {X 0,Y 112.877,Z 589.602,A -85,B 0,C 180,E1 -28230.651,E2 -28230.651} C_VEL
LIN {X 0,Y 122.911,Z 580.319,A -85,B 0,C 180,E1 -28234.231,E2 -28234.231} C_VEL
LIN {X 0,Y 131.812,Z 570.889,A -85,B 0,C 180,E1 -28236.885,E2 -28236.885} C_VEL
LIN {X 0,Y 141.316,Z 559.31,A -85,B 0,C 180,E1 -28239.189,E2 -28239.189} C_VEL
LIN {X 0,Y 144.263,Z 554.893,A -85,B 0,C 180,E1 -28240.211,E2 -28240.211} C_VEL
LIN {X 0,Y 151.318,Z 541.518,A -85,B 0,C 180,E1 -28243.863,E2 -28243.863} C_VEL
LIN {X 0,Y 153.885,Z 536.649,A -85,B 0,C 180,E1 -28244.689,E2 -28244.689} C_VEL
LIN {X 0,Y 154.826,Z 534.961,A -85,B 0,C 180,E1 -28244.863,E2 -28244.863} C_VEL
LIN {X 0,Y 162.093,Z 520.451,A -85,B 0,C 180,E1 -28245.954,E2 -28245.954} C_VEL
LIN {X 0,Y 167.889,Z 505.93,A -85,B 0,C 180,E1 -28246.716,E2 -28246.716} C_VEL
LIN {X 0,Y 172.434,Z 490.856,A -85,B 0,C 180,E1 -28247.318,E2 -28247.318} C_VEL
LIN {X 0,Y 175.715,Z 475.25,A -85,B 0,C 180,E1 -28247.739,E2 -28247.739} C_VEL
LIN {X 0,Y 178.815,Z 449.85,A -85,B 0,C 180,E1 -28248.254,E2 -28248.254} C_VEL
LIN {X 0,Y 177.333,Z 445.529,A -85,B 0,C 180,E1 -28251.884,E2 -28251.884} C_VEL
LIN {X 0,Y 176.664,Z 443.406,A -85,B 0,C 180,E1 -28254.293,E2 -28254.293} C_VEL
LIN {X 0,Y 176.113,Z 440.429,A -85,B 0,C 180,E1 -28259.187,E2 -28259.187} C_VEL
LIN {X 0,Y 176.116,Z 440.565,A -85,B 0,C 180,E1 -28261.572,E2 -28261.572} C_VEL
LIN {X 0,Y 176.944,Z 444.323,A -85,B 0,C 180,E1 -28267.274,E2 -28267.274} C_VEL
LIN {X 0,Y 177.999,Z 447.543,A -85,B 0,C 180,E1 -28270.378,E2 -28270.378} C_VEL
LIN {X 0,Y 178.781,Z 449.768,A -85,B 0,C 180,E1 -28272.126,E2 -28272.126} C_VEL
LIN {X 0,Y 175.77,Z 473.988,A -85,B 0,C 180,E1 -28272.649,E2 -28272.649} C_VEL
LIN {X 0,Y 172.849,Z 488.075,A -85,B 0,C 180,E1 -28273.08,E2 -28273.08} C_VEL
LIN {X 0,Y 168.234,Z 503.602,A -85,B 0,C 180,E1 -28273.773,E2 -28273.773} C_VEL
LIN {X 0,Y 162.533,Z 518.087,A -85,B 0,C 180,E1 -28274.652,E2 -28274.652} C_VEL
LIN {X 0,Y 155.779,Z 531.845,A -85,B 0,C 180,E1 -28275.816,E2 -28275.816} C_VEL
LIN {X 0,Y 148.134,Z 544.719,A -85,B 0,C 180,E1 -28277.298,E2 -28277.298} C_VEL
LIN {X 0,Y 139.411,Z 556.914,A -85,B 0,C 180,E1 -28279.056,E2 -28279.056} C_VEL
LIN {X 0,Y 130.109,Z 568.021,A -85,B 0,C 180,E1 -28281.29,E2 -28281.29} C_VEL
LIN {X 0,Y 119.543,Z 578.73,A -85,B 0,C 180,E1 -28284.211,E2 -28284.211} C_VEL
LIN {X 0,Y 109.387,Z 587.746,A -85,B 0,C 180,E1 -28287.945,E2 -28287.945} C_VEL
LIN {X 0,Y 99.635,Z 595.16,A -85,B 0,C 180,E1 -28292.175,E2 -28292.175} C_VEL
LIN {X 0,Y 89.289,Z 602.081,A -85,B 0,C 180,E1 -28298.086,E2 -28298.086} C_VEL
LIN {X 0,Y 80.145,Z 607.507,A -85,B 0,C 180,E1 -28305.452,E2 -28305.452} C_VEL
LIN {X 0,Y 72.489,Z 611.595,A -85,B 0,C 180,E1 -28314.43,E2 -28314.43} C_VEL
LIN {X 0,Y 66.904,Z 614.453,A -85,B 0,C 180,E1 -28325.155,E2 -28325.155} C_VEL
LIN {X 0,Y 63.597,Z 616.161,A -85,B 0,C 180,E1 -28337.232,E2 -28337.232} C_VEL
LIN {X 0,Y 62.699,Z 616.748,A -85,B 0,C 180,E1 -28350,E2 -28350} C_VEL
LIN {X 0,Y 63.593,Z 616.19,A -85,B 0,C 180,E1 -28362.769,E2 -28362.769} C_VEL
LIN {X 0,Y 66.826,Z 614.521,A -85,B 0,C 180,E1 -28374.877,E2 -28374.877} C_VEL
LIN {X 0,Y 72.458,Z 611.695,A -85,B 0,C 180,E1 -28385.588,E2 -28385.588} C_VEL
LIN {X 0,Y 80.118,Z 607.638,A -85,B 0,C 180,E1 -28394.568,E2 -28394.568} C_VEL
LIN {X 0,Y 89.258,Z 602.254,A -85,B 0,C 180,E1 -28401.939,E2 -28401.939} C_VEL
LIN {X 0,Y 99.585,Z 595.383,A -85,B 0,C 180,E1 -28407.871,E2 -28407.871} C_VEL
LIN {X 0,Y 109.349,Z 587.995,A -85,B 0,C 180,E1 -28412.093,E2 -28412.093} C_VEL
LIN {X 0,Y 119.41,Z 579.096,A -85,B 0,C 180,E1 -28415.814,E2 -28415.814} C_VEL
LIN {X 0,Y 128.514,Z 569.997,A -85,B 0,C 180,E1 -28418.38,E2 -28418.38} C_VEL
LIN {X 0,Y 137.814,Z 559.265,A -85,B 0,C 180,E1 -28420.631,E2 -28420.631} C_VEL
LIN {X 0,Y 146.485,Z 547.544,A -85,B 0,C 180,E1 -28422.464,E2 -28422.464} C_VEL
LIN {X 0,Y 154.936,Z 533.904,A -85,B 0,C 180,E1 -28424.059,E2 -28424.059} C_VEL
LIN {X 0,Y 161.69,Z 520.596,A -85,B 0,C 180,E1 -28425.26,E2 -28425.26} C_VEL
LIN {X 0,Y 167.365,Z 506.794,A -85,B 0,C 180,E1 -28426.177,E2 -28426.177} C_VEL
LIN {X 0,Y 172.267,Z 491.326,A -85,B 0,C 180,E1 -28426.907,E2 -28426.907} C_VEL
LIN {X 0,Y 175.6,Z 476.534,A -85,B 0,C 180,E1 -28427.41,E2 -28427.41} C_VEL
LIN {X 0,Y 178.14,Z 458.19,A -85,B 0,C 180,E1 -28427.809,E2 -28427.809} C_VEL
LIN {X 0,Y 179.043,Z 449.99,A -85,B 0,C 180,E1 -28428,E2 -28428} C_VEL
LIN {X 0,Y 177.656,Z 445.916,A -85,B 0,C 180,E1 -28431.412,E2 -28431.412} C_VEL
LIN {X 0,Y 176.906,Z 443.595,A -85,B 0,C 180,E1 -28434.12,E2 -28434.12} C_VEL
LIN {X 0,Y 176.411,Z 440.531,A -85,B 0,C 180,E1 -28439.429,E2 -28439.429} C_VEL
LIN {X 0,Y 176.407,Z 440.763,A -85,B 0,C 180,E1 -28440.856,E2 -28440.856} C_VEL
LIN {X 0,Y 177.16,Z 444.33,A -85,B 0,C 180,E1 -28446.549,E2 -28446.549} C_VEL
LIN {X 0,Y 178.274,Z 447.743,A -85,B 0,C 180,E1 -28449.902,E2 -28449.902} C_VEL
LIN {X 0,Y 179.066,Z 450.032,A -85,B 0,C 180,E1 -28451.687,E2 -28451.687} C_VEL
LIN {X 0,Y 176.076,Z 474.827,A -85,B 0,C 180,E1 -28452.209,E2 -28452.209} C_VEL
LIN {X 0,Y 172.852,Z 490.37,A -85,B 0,C 180,E1 -28452.633,E2 -28452.633} C_VEL
LIN {X 0,Y 168.304,Z 505.571,A -85,B 0,C 180,E1 -28453.232,E2 -28453.232} C_VEL
LIN {X 0,Y 162.918,Z 519.281,A -85,B 0,C 180,E1 -28453.932,E2 -28453.932} C_VEL
LIN {X 0,Y 156.374,Z 532.719,A -85,B 0,C 180,E1 -28454.926,E2 -28454.926} C_VEL
LIN {X 0,Y 149.027,Z 545.111,A -85,B 0,C 180,E1 -28456.087,E2 -28456.087} C_VEL
LIN {X 0,Y 141.425,Z 556.138,A -85,B 0,C 180,E1 -28457.557,E2 -28457.557} C_VEL
LIN {X 0,Y 132.335,Z 567.42,A -85,B 0,C 180,E1 -28459.501,E2 -28459.501} C_VEL
LIN {X 0,Y 123.025,Z 577.378,A -85,B 0,C 180,E1 -28461.831,E2 -28461.831} C_VEL
LIN {X 0,Y 112.478,Z 587.127,A -85,B 0,C 180,E1 -28465.044,E2 -28465.044} C_VEL
LIN {X 0,Y 102.459,Z 595.273,A -85,B 0,C 180,E1 -28469.01,E2 -28469.01} C_VEL
LIN {X 0,Y 93.054,Z 602.02,A -85,B 0,C 180,E1 -28473.823,E2 -28473.823} C_VEL
LIN {X 0,Y 83.148,Z 608.249,A -85,B 0,C 180,E1 -28480.475,E2 -28480.475} C_VEL
LIN {X 0,Y 74.737,Z 613.079,A -85,B 0,C 180,E1 -28488.835,E2 -28488.835} C_VEL
LIN {X 0,Y 68.204,Z 616.628,A -85,B 0,C 180,E1 -28498.989,E2 -28498.989} C_VEL
LIN {X 0,Y 64.004,Z 618.974,A -85,B 0,C 180,E1 -28510.767,E2 -28510.767} C_VEL
LIN {X 0,Y 62.45,Z 620.166,A -85,B 0,C 180,E1 -28523.538,E2 -28523.538} C_VEL
LIN {X 0,Y 62.555,Z 620.33,A -85,B 0,C 180,E1 -28530,E2 -28530} C_VEL
LIN {X 0,Y 62.882,Z 619.69,A -85,B 0,C 180,E1 -28542.916,E2 -28542.916} C_VEL
LIN {X 0,Y 65.707,Z 617.894,A -85,B 0,C 180,E1 -28555.33,E2 -28555.33} C_VEL
LIN {X 0,Y 71.133,Z 614.93,A -85,B 0,C 180,E1 -28566.355,E2 -28566.355} C_VEL
LIN {X 0,Y 78.717,Z 610.731,A -85,B 0,C 180,E1 -28575.58,E2 -28575.58} C_VEL
LIN {X 0,Y 87.936,Z 605.186,A -85,B 0,C 180,E1 -28583.053,E2 -28583.053} C_VEL
LIN {X 0,Y 98.359,Z 598.147,A -85,B 0,C 180,E1 -28589.026,E2 -28589.026} C_VEL
LIN {X 0,Y 108.095,Z 590.624,A -85,B 0,C 180,E1 -28593.373,E2 -28593.373} C_VEL
LIN {X 0,Y 118.459,Z 581.567,A -85,B 0,C 180,E1 -28596.863,E2 -28596.863} C_VEL
LIN {X 0,Y 129.182,Z 570.683,A -85,B 0,C 180,E1 -28599.791,E2 -28599.791} C_VEL
LIN {X 0,Y 138.643,Z 559.487,A -85,B 0,C 180,E1 -28601.885,E2 -28601.885} C_VEL
LIN {X 0,Y 147.414,Z 547.211,A -85,B 0,C 180,E1 -28603.625,E2 -28603.625} C_VEL
LIN {X 0,Y 154.826,Z 534.961,A -85,B 0,C 180,E1 -28604.863,E2 -28604.863} C_VEL
LIN {X 0,Y 157.405,Z 529.942,A -85,B 0,C 180,E1 -28605.504,E2 -28605.504} C_VEL
LIN {X 0,Y 160.733,Z 521.679,A -85,B 0,C 180,E1 -28607.073,E2 -28607.073} C_VEL
LIN {X 0,Y 163.723,Z 513.169,A -85,B 0,C 180,E1 -28608.522,E2 -28608.522} C_VEL
LIN {X 0,Y 165.637,Z 507.764,A -85,B 0,C 180,E1 -28609.012,E2 -28609.012} C_VEL
LIN {X 0,Y 170.391,Z 492.933,A -85,B 0,C 180,E1 -28609.559,E2 -28609.559} C_VEL
LIN {X 0,Y 173.952,Z 477.198,A -85,B 0,C 180,E1 -28609.967,E2 -28609.967} C_VEL
LIN {X 0,Y 176.766,Z 456.081,A -85,B 0,C 180,E1 -28610.378,E2 -28610.378} C_VEL
LIN {X 0,Y 176.92,Z 454.576,A -85,B 0,C 180,E1 -28610.44,E2 -28610.44} C_VEL
LIN {X 0,Y 175.884,Z 451.07,A -85,B 0,C 180,E1 -28613.792,E2 -28613.792} C_VEL
LIN {X 0,Y 175.241,Z 447.532,A -85,B 0,C 180,E1 -28619.183,E2 -28619.183} C_VEL
LIN {X 0,Y 175.232,Z 447.617,A -85,B 0,C 180,E1 -28621.293,E2 -28621.293} C_VEL
LIN {X 0,Y 175.868,Z 451.039,A -85,B 0,C 180,E1 -28626.598,E2 -28626.598} C_VEL
LIN {X 0,Y 176.916,Z 454.525,A -85,B 0,C 180,E1 -28629.988,E2 -28629.988} C_VEL
LIN {X 0,Y 174.182,Z 475.182,A -85,B 0,C 180,E1 -28630.409,E2 -28630.409} C_VEL
LIN {X 0,Y 171.333,Z 488.48,A -85,B 0,C 180,E1 -28630.78,E2 -28630.78} C_VEL
LIN {X 0,Y 167.067,Z 502.787,A -85,B 0,C 180,E1 -28631.365,E2 -28631.365} C_VEL
LIN {X 0,Y 161.712,Z 516.445,A -85,B 0,C 180,E1 -28632.089,E2 -28632.089} C_VEL
LIN {X 0,Y 155.014,Z 530.178,A -85,B 0,C 180,E1 -28633.103,E2 -28633.103} C_VEL
LIN {X 0,Y 146.989,Z 543.692,A -85,B 0,C 180,E1 -28634.49,E2 -28634.49} C_VEL
LIN {X 0,Y 138.871,Z 555.023,A -85,B 0,C 180,E1 -28635.945,E2 -28635.945} C_VEL
LIN {X 0,Y 129.302,Z 566.462,A -85,B 0,C 180,E1 -28637.981,E2 -28637.981} C_VEL
LIN {X 0,Y 119.821,Z 576.092,A -85,B 0,C 180,E1 -28640.209,E2 -28640.209} C_VEL
LIN {X 0,Y 112.18,Z 583.041,A -85,B 0,C 180,E1 -28642.475,E2 -28642.475} C_VEL
LIN {X 0,Y 103.241,Z 590.176,A -85,B 0,C 180,E1 -28645.584,E2 -28645.584} C_VEL
LIN {X 0,Y 93.207,Z 597.229,A -85,B 0,C 180,E1 -28649.877,E2 -28649.877} C_VEL
LIN {X 0,Y 82.509,Z 603.765,A -85,B 0,C 180,E1 -28655.985,E2 -28655.985} C_VEL
LIN {X 0,Y 72.965,Z 608.865,A -85,B 0,C 180,E1 -28663.749,E2 -28663.749} C_VEL
LIN {X 0,Y 66.828,Z 611.799,A -85,B 0,C 180,E1 -28670.878,E2 -28670.878} C_VEL
LIN {X 0,Y 60.495,Z 614.658,A -85,B 0,C 180,E1 -28682.31,E2 -28682.31} C_VEL
LIN {X 0,Y 56.681,Z 616.365,A -85,B 0,C 180,E1 -28695.642,E2 -28695.642} C_VEL
LIN {X 0,Y 55.608,Z 616.951,A -85,B 0,C 180,E1 -28710,E2 -28710} C_VEL
LIN {X 0,Y 56.676,Z 616.393,A -85,B 0,C 180,E1 -28724.359,E2 -28724.359} C_VEL
LIN {X 0,Y 60.424,Z 614.725,A -85,B 0,C 180,E1 -28737.725,E2 -28737.725} C_VEL
LIN {X 0,Y 66.801,Z 611.897,A -85,B 0,C 180,E1 -28749.141,E2 -28749.141} C_VEL
LIN {X 0,Y 75.202,Z 607.841,A -85,B 0,C 180,E1 -28758.385,E2 -28758.385} C_VEL
LIN {X 0,Y 85.041,Z 602.456,A -85,B 0,C 180,E1 -28765.731,E2 -28765.731} C_VEL
LIN {X 0,Y 95.975,Z 595.586,A -85,B 0,C 180,E1 -28771.487,E2 -28771.487} C_VEL
LIN {X 0,Y 106.2,Z 588.197,A -85,B 0,C 180,E1 -28775.493,E2 -28775.493} C_VEL
LIN {X 0,Y 116.677,Z 579.297,A -85,B 0,C 180,E1 -28779,E2 -28779} C_VEL
LIN {X 0,Y 126.072,Z 570.197,A -85,B 0,C 180,E1 -28781.38,E2 -28781.38} C_VEL
LIN {X 0,Y 135.619,Z 559.465,A -85,B 0,C 180,E1 -28783.471,E2 -28783.471} C_VEL
LIN {X 0,Y 144.507,Z 547.743,A -85,B 0,C 180,E1 -28785.145,E2 -28785.145} C_VEL
LIN {X 0,Y 153.132,Z 534.103,A -85,B 0,C 180,E1 -28786.623,E2 -28786.623} C_VEL
LIN {X 0,Y 160.032,Z 520.793,A -85,B 0,C 180,E1 -28787.717,E2 -28787.717} C_VEL
LIN {X 0,Y 165.814,Z 506.99,A -85,B 0,C 180,E1 -28788.557,E2 -28788.557} C_VEL
LIN {X 0,Y 170.801,Z 491.519,A -85,B 0,C 180,E1 -28789.224,E2 -28789.224} C_VEL
LIN {X 0,Y 174.248,Z 476.425,A -85,B 0,C 180,E1 -28789.69,E2 -28789.69} C_VEL
LIN {X 0,Y 176.751,Z 458.624,A -85,B 0,C 180,E1 -28790.047,E2 -28790.047} C_VEL
LIN {X 0,Y 177.174,Z 454.704,A -85,B 0,C 180,E1 -28790.171,E2 -28790.171} C_VEL
LIN {X 0,Y 176.073,Z 450.926,A -85,B 0,C 180,E1 -28793.891,E2 -28793.891} C_VEL
LIN {X 0,Y 175.541,Z 447.622,A -85,B 0,C 180,E1 -28799.426,E2 -28799.426} C_VEL
LIN {X 0,Y 175.524,Z 447.961,A -85,B 0,C 180,E1 -28800.86,E2 -28800.86} C_VEL
LIN {X 0,Y 176.125,Z 451.194,A -85,B 0,C 180,E1 -28806.012,E2 -28806.012} C_VEL
LIN {X 0,Y 177.142,Z 454.614,A -85,B 0,C 180,E1 -28809.39,E2 -28809.39} C_VEL
LIN {X 0,Y 177.189,Z 454.791,A -85,B 0,C 180,E1 -28809.521,E2 -28809.521} C_VEL
LIN {X 0,Y 174.646,Z 474.999,A -85,B 0,C 180,E1 -28809.942,E2 -28809.942} C_VEL
LIN {X 0,Y 171.309,Z 490.643,A -85,B 0,C 180,E1 -28810.329,E2 -28810.329} C_VEL
LIN {X 0,Y 166.824,Z 505.376,A -85,B 0,C 180,E1 -28810.862,E2 -28810.862} C_VEL
LIN {X 0,Y 161.357,Z 519.084,A -85,B 0,C 180,E1 -28811.486,E2 -28811.486} C_VEL
LIN {X 0,Y 154.692,Z 532.521,A -85,B 0,C 180,E1 -28812.375,E2 -28812.375} C_VEL
LIN {X 0,Y 147.208,Z 544.911,A -85,B 0,C 180,E1 -28813.415,E2 -28813.415} C_VEL
LIN {X 0,Y 138.226,Z 557.536,A -85,B 0,C 180,E1 -28814.981,E2 -28814.981} C_VEL
LIN {X 0,Y 128.523,Z 569.009,A -85,B 0,C 180,E1 -28816.878,E2 -28816.878} C_VEL
LIN {X 0,Y 118.974,Z 578.668,A -85,B 0,C 180,E1 -28819.07,E2 -28819.07} C_VEL
LIN {X 0,Y 108.113,Z 588.163,A -85,B 0,C 180,E1 -28822.133,E2 -28822.133} C_VEL
LIN {X 0,Y 97.733,Z 596.086,A -85,B 0,C 180,E1 -28825.993,E2 -28825.993} C_VEL
LIN {X 0,Y 86.506,Z 603.489,A -85,B 0,C 180,E1 -28831.457,E2 -28831.457} C_VEL
LIN {X 0,Y 76.245,Z 609.368,A -85,B 0,C 180,E1 -28838.42,E2 -28838.42} C_VEL
LIN {X 0,Y 69.052,Z 613.102,A -85,B 0,C 180,E1 -28845.434,E2 -28845.434} C_VEL
LIN {X 0,Y 62.169,Z 616.424,A -85,B 0,C 180,E1 -28855.582,E2 -28855.582} C_VEL
LIN {X 0,Y 57.291,Z 618.769,A -85,B 0,C 180,E1 -28868.407,E2 -28868.407} C_VEL
LIN {X 0,Y 55.369,Z 619.962,A -85,B 0,C 180,E1 -28882.708,E2 -28882.708} C_VEL
LIN {X 0,Y 55.463,Z 620.127,A -85,B 0,C 180,E1 -28890,E2 -28890} C_VEL
LIN {X 0,Y 55.956,Z 619.486,A -85,B 0,C 180,E1 -28904.548,E2 -28904.548} C_VEL
LIN {X 0,Y 59.315,Z 617.689,A -85,B 0,C 180,E1 -28918.29,E2 -28918.29} C_VEL
LIN {X 0,Y 65.483,Z 614.724,A -85,B 0,C 180,E1 -28930.086,E2 -28930.086} C_VEL
LIN {X 0,Y 73.868,Z 610.525,A -85,B 0,C 180,E1 -28939.563,E2 -28939.563} C_VEL
LIN {X 0,Y 83.822,Z 604.98,A -85,B 0,C 180,E1 -28946.973,E2 -28946.973} C_VEL
LIN {X 0,Y 94.862,Z 597.94,A -85,B 0,C 180,E1 -28952.749,E2 -28952.749} C_VEL
LIN {X 0,Y 105.074,Z 590.417,A -85,B 0,C 180,E1 -28956.873,E2 -28956.873} C_VEL
LIN {X 0,Y 115.843,Z 581.361,A -85,B 0,C 180,E1 -28960.107,E2 -28960.107} C_VEL
LIN {X 0,Y 126.899,Z 570.477,A -85,B 0,C 180,E1 -28962.808,E2 -28962.808} C_VEL
LIN {X 0,Y 137.401,Z 558.242,A -85,B 0,C 180,E1 -28964.888,E2 -28964.888} C_VEL
LIN {X 0,Y 146.386,Z 545.765,A -85,B 0,C 180,E1 -28966.452,E2 -28966.452} C_VEL
LIN {X 0,Y 153.852,Z 533.508,A -85,B 0,C 180,E1 -28967.525,E2 -28967.525} C_VEL
LIN {X 0,Y 160.518,Z 520.242,A -85,B 0,C 180,E1 -28968.414,E2 -28968.414} C_VEL
LIN {X 0,Y 165.637,Z 507.764,A -85,B 0,C 180,E1 -28969.012,E2 -28969.012} C_VEL
LIN {X 0,Y 167.465,Z 502.296,A -85,B 0,C 180,E1 -28969.452,E2 -28969.452} C_VEL
LIN {X 0,Y 169.703,Z 493.373,A -85,B 0,C 180,E1 -28970.704,E2 -28970.704} C_VEL
LIN {X 0,Y 171.507,Z 484.298,A -85,B 0,C 180,E1 -28971.893,E2 -28971.893} C_VEL
LIN {X 0,Y 172.554,Z 478.59,A -85,B 0,C 180,E1 -28972.259,E2 -28972.259} C_VEL
LIN {X 0,Y 175.212,Z 460.15,A -85,B 0,C 180,E1 -28972.598,E2 -28972.598} C_VEL
LIN {X 0,Y 175.27,Z 459.475,A -85,B 0,C 180,E1 -28972.661,E2 -28972.661} C_VEL
LIN {X 0,Y 174.657,Z 457.121,A -85,B 0,C 180,E1 -28975.384,E2 -28975.384} C_VEL
LIN {X 0,Y 174.364,Z 454.445,A -85,B 0,C 180,E1 -28980,E2 -28980} C_VEL
LIN {X 0,Y 174.336,Z 455.125,A -85,B 0,C 180,E1 -28981.681,E2 -28981.681} C_VEL
LIN {X 0,Y 174.845,Z 457.894,A -85,B 0,C 180,E1 -28986.057,E2 -28986.057} C_VEL
LIN {X 0,Y 175.261,Z 459.494,A -85,B 0,C 180,E1 -28987.769,E2 -28987.769} C_VEL
LIN {X 0,Y 172.855,Z 476.405,A -85,B 0,C 180,E1 -28988.122,E2 -28988.122} C_VEL
LIN {X 0,Y 169.662,Z 490.469,A -85,B 0,C 180,E1 -28988.506,E2 -28988.506} C_VEL
LIN {X 0,Y 164.882,Z 505.492,A -85,B 0,C 180,E1 -28989.065,E2 -28989.065} C_VEL
LIN {X 0,Y 159.535,Z 518.504,A -85,B 0,C 180,E1 -28989.715,E2 -28989.715} C_VEL
LIN {X 0,Y 152.522,Z 532.26,A -85,B 0,C 180,E1 -28990.676,E2 -28990.676} C_VEL
LIN {X 0,Y 144.547,Z 545.133,A -85,B 0,C 180,E1 -28991.912,E2 -28991.912} C_VEL
LIN {X 0,Y 135.445,Z 557.326,A -85,B 0,C 180,E1 -28993.375,E2 -28993.375} C_VEL
LIN {X 0,Y 125.656,Z 568.432,A -85,B 0,C 180,E1 -28995.252,E2 -28995.252} C_VEL
LIN {X 0,Y 115.954,Z 577.776,A -85,B 0,C 180,E1 -28997.337,E2 -28997.337} C_VEL
LIN {X 0,Y 106.567,Z 585.723,A -85,B 0,C 180,E1 -28999.991,E2 -28999.991} C_VEL
LIN {X 0,Y 95.808,Z 593.572,A -85,B 0,C 180,E1 -29003.521,E2 -29003.521} C_VEL
LIN {X 0,Y 84.088,Z 600.892,A -85,B 0,C 180,E1 -29008.652,E2 -29008.652} C_VEL
LIN {X 0,Y 74.121,Z 606.265,A -85,B 0,C 180,E1 -29014.675,E2 -29014.675} C_VEL
LIN {X 0,Y 65.897,Z 610.119,A -85,B 0,C 180,E1 -29021.708,E2 -29021.708} C_VEL
LIN {X 0,Y 57.529,Z 613.582,A -85,B 0,C 180,E1 -29032.352,E2 -29032.352} C_VEL
LIN {X 0,Y 51.681,Z 615.856,A -85,B 0,C 180,E1 -29045.924,E2 -29045.924} C_VEL
LIN {X 0,Y 48.804,Z 617.003,A -85,B 0,C 180,E1 -29061.721,E2 -29061.721} C_VEL
LIN {X 0,Y 48.508,Z 617.154,A -85,B 0,C 180,E1 -29070,E2 -29070} C_VEL
LIN {X 0,Y 49.827,Z 616.596,A -85,B 0,C 180,E1 -29086.385,E2 -29086.385} C_VEL
LIN {X 0,Y 54.214,Z 614.928,A -85,B 0,C 180,E1 -29101.233,E2 -29101.233} C_VEL
LIN {X 0,Y 61.448,Z 612.1,A -85,B 0,C 180,E1 -29113.331,E2 -29113.331} C_VEL
LIN {X 0,Y 70.667,Z 608.044,A -85,B 0,C 180,E1 -29122.712,E2 -29122.712} C_VEL
LIN {X 0,Y 81.232,Z 602.659,A -85,B 0,C 180,E1 -29129.9,E2 -29129.9} C_VEL
LIN {X 0,Y 92.777,Z 595.789,A -85,B 0,C 180,E1 -29135.366,E2 -29135.366} C_VEL
LIN {X 0,Y 103.441,Z 588.4,A -85,B 0,C 180,E1 -29139.096,E2 -29139.096} C_VEL
LIN {X 0,Y 114.318,Z 579.498,A -85,B 0,C 180,E1 -29142.334,E2 -29142.334} C_VEL
LIN {X 0,Y 123.983,Z 570.398,A -85,B 0,C 180,E1 -29144.498,E2 -29144.498} C_VEL
LIN {X 0,Y 133.767,Z 559.666,A -85,B 0,C 180,E1 -29146.396,E2 -29146.396} C_VEL
LIN {X 0,Y 142.853,Z 547.942,A -85,B 0,C 180,E1 -29147.896,E2 -29147.896} C_VEL
LIN {X 0,Y 151.265,Z 534.952,A -85,B 0,C 180,E1 -29149.179,E2 -29149.179} C_VEL
LIN {X 0,Y 157.836,Z 522.751,A -85,B 0,C 180,E1 -29150.109,E2 -29150.109} C_VEL
LIN {X 0,Y 163.712,Z 509.44,A -85,B 0,C 180,E1 -29150.874,E2 -29150.874} C_VEL
LIN {X 0,Y 168.487,Z 495.73,A -85,B 0,C 180,E1 -29151.446,E2 -29151.446} C_VEL
LIN {X 0,Y 172.361,Z 480.625,A -85,B 0,C 180,E1 -29151.895,E2 -29151.895} C_VEL
LIN {X 0,Y 174.861,Z 465.598,A -85,B 0,C 180,E1 -29152.192,E2 -29152.192} C_VEL
LIN {X 0,Y 175.534,Z 459.664,A -85,B 0,C 180,E1 -29152.385,E2 -29152.385} C_VEL
LIN {X 0,Y 174.936,Z 457.339,A -85,B 0,C 180,E1 -29155.102,E2 -29155.102} C_VEL
LIN {X 0,Y 174.676,Z 454.637,A -85,B 0,C 180,E1 -29160,E2 -29160} C_VEL
LIN {X 0,Y 175.109,Z 458.026,A -85,B 0,C 180,E1 -29165.47,E2 -29165.47} C_VEL
LIN {X 0,Y 175.559,Z 459.716,A -85,B 0,C 180,E1 -29167.334,E2 -29167.334} C_VEL
LIN {X 0,Y 173.307,Z 476.178,A -85,B 0,C 180,E1 -29167.661,E2 -29167.661} C_VEL
LIN {X 0,Y 169.89,Z 491.492,A -85,B 0,C 180,E1 -29168.009,E2 -29168.009} C_VEL
LIN {X 0,Y 165.138,Z 506.483,A -85,B 0,C 180,E1 -29168.487,E2 -29168.487} C_VEL
LIN {X 0,Y 159.242,Z 520.672,A -85,B 0,C 180,E1 -29169.079,E2 -29169.079} C_VEL
LIN {X 0,Y 152.479,Z 533.812,A -85,B 0,C 180,E1 -29169.877,E2 -29169.877} C_VEL
LIN {X 0,Y 144.043,Z 547.203,A -85,B 0,C 180,E1 -29170.921,E2 -29170.921} C_VEL
LIN {X 0,Y 134.895,Z 559.413,A -85,B 0,C 180,E1 -29172.355,E2 -29172.355} C_VEL
LIN {X 0,Y 124.99,Z 570.565,A -85,B 0,C 180,E1 -29174.091,E2 -29174.091} C_VEL
LIN {X 0,Y 115.216,Z 579.958,A -85,B 0,C 180,E1 -29176.117,E2 -29176.117} C_VEL
LIN {X 0,Y 104.049,Z 589.2,A -85,B 0,C 180,E1 -29178.985,E2 -29178.985} C_VEL
LIN {X 0,Y 94.444,Z 596.122,A -85,B 0,C 180,E1 -29182.217,E2 -29182.217} C_VEL
LIN {X 0,Y 82.991,Z 603.285,A -85,B 0,C 180,E1 -29187.233,E2 -29187.233} C_VEL
LIN {X 0,Y 72.004,Z 609.164,A -85,B 0,C 180,E1 -29193.939,E2 -29193.939} C_VEL
LIN {X 0,Y 63.485,Z 613.204,A -85,B 0,C 180,E1 -29201.621,E2 -29201.621} C_VEL
LIN {X 0,Y 56.391,Z 616.219,A -85,B 0,C 180,E1 -29211.455,E2 -29211.455} C_VEL
LIN {X 0,Y 50.691,Z 618.565,A -85,B 0,C 180,E1 -29225.423,E2 -29225.423} C_VEL
LIN {X 0,Y 48.319,Z 619.759,A -85,B 0,C 180,E1 -29241.637,E2 -29241.637} C_VEL
LIN {X 0,Y 48.355,Z 619.924,A -85,B 0,C 180,E1 -29250,E2 -29250} C_VEL
LIN {X 0,Y 49.065,Z 619.281,A -85,B 0,C 180,E1 -29266.646,E2 -29266.646} C_VEL
LIN {X 0,Y 53.124,Z 617.484,A -85,B 0,C 180,E1 -29281.949,E2 -29281.949} C_VEL
LIN {X 0,Y 60.168,Z 614.518,A -85,B 0,C 180,E1 -29294.493,E2 -29294.493} C_VEL
LIN {X 0,Y 69.443,Z 610.319,A -85,B 0,C 180,E1 -29304.059,E2 -29304.059} C_VEL
LIN {X 0,Y 80.14,Z 604.773,A -85,B 0,C 180,E1 -29311.276,E2 -29311.276} C_VEL
LIN {X 0,Y 91.805,Z 597.734,A -85,B 0,C 180,E1 -29316.725,E2 -29316.725} C_VEL
LIN {X 0,Y 102.478,Z 590.209,A -85,B 0,C 180,E1 -29320.554,E2 -29320.554} C_VEL
LIN {X 0,Y 113.606,Z 581.154,A -85,B 0,C 180,E1 -29323.506,E2 -29323.506} C_VEL
LIN {X 0,Y 123.333,Z 571.911,A -85,B 0,C 180,E1 -29325.627,E2 -29325.627} C_VEL
LIN {X 0,Y 133.237,Z 561.031,A -85,B 0,C 180,E1 -29327.371,E2 -29327.371} C_VEL
LIN {X 0,Y 142.491,Z 548.982,A -85,B 0,C 180,E1 -29328.852,E2 -29328.852} C_VEL
LIN {X 0,Y 150.78,Z 536.16,A -85,B 0,C 180,E1 -29329.941,E2 -29329.941} C_VEL
LIN {X 0,Y 158.394,Z 521.802,A -85,B 0,C 180,E1 -29330.827,E2 -29330.827} C_VEL
LIN {X 0,Y 164.284,Z 507.946,A -85,B 0,C 180,E1 -29331.427,E2 -29331.427} C_VEL
LIN {X 0,Y 169.135,Z 493.123,A -85,B 0,C 180,E1 -29331.913,E2 -29331.913} C_VEL
LIN {X 0,Y 172.554,Z 478.59,A -85,B 0,C 180,E1 -29332.259,E2 -29332.259} C_VEL
LIN {X 0,Y 173.191,Z 474.586,A -85,B 0,C 180,E1 -29332.598,E2 -29332.598} C_VEL
LIN {X 0,Y 173.503,Z 470.95,A -85,B 0,C 180,E1 -29333.299,E2 -29333.299} C_VEL
LIN {X 0,Y 173.646,Z 466.899,A -85,B 0,C 180,E1 -29334.614,E2 -29334.614} C_VEL
LIN {X 0,Y 173.632,Z 464.619,A -85,B 0,C 180,E1 -29335.811,E2 -29335.811} C_VEL
LIN {X 0,Y 173.532,Z 463.255,A -85,B 0,C 180,E1 -29337.144,E2 -29337.144} C_VEL
LIN {X 0,Y 173.497,Z 461.513,A -85,B 0,C 180,E1 -29340,E2 -29340} C_VEL
LIN {X 0,Y 173.463,Z 462.72,A -85,B 0,C 180,E1 -29342.322,E2 -29342.322} C_VEL
LIN {X 0,Y 173.841,Z 464.772,A -85,B 0,C 180,E1 -29345.532,E2 -29345.532} C_VEL
LIN {X 0,Y 171.311,Z 480.226,A -85,B 0,C 180,E1 -29345.834,E2 -29345.834} C_VEL
LIN {X 0,Y 167.267,Z 495.931,A -85,B 0,C 180,E1 -29346.278,E2 -29346.278} C_VEL
LIN {X 0,Y 161.906,Z 510.921,A -85,B 0,C 180,E1 -29346.82,E2 -29346.82} C_VEL
LIN {X 0,Y 155.19,Z 525.467,A -85,B 0,C 180,E1 -29347.585,E2 -29347.585} C_VEL
LIN {X 0,Y 148.317,Z 537.606,A -85,B 0,C 180,E1 -29348.456,E2 -29348.456} C_VEL
LIN {X 0,Y 139.024,Z 551.171,A -85,B 0,C 180,E1 -29349.686,E2 -29349.686} C_VEL
LIN {X 0,Y 128.967,Z 563.328,A -85,B 0,C 180,E1 -29351.223,E2 -29351.223} C_VEL
LIN {X 0,Y 118.976,Z 573.508,A -85,B 0,C 180,E1 -29352.931,E2 -29352.931} C_VEL
LIN {X 0,Y 108.093,Z 582.976,A -85,B 0,C 180,E1 -29355.249,E2 -29355.249} C_VEL
LIN {X 0,Y 97.948,Z 590.586,A -85,B 0,C 180,E1 -29358.068,E2 -29358.068} C_VEL
LIN {X 0,Y 86.99,Z 597.639,A -85,B 0,C 180,E1 -29361.711,E2 -29361.711} C_VEL
LIN {X 0,Y 75.014,Z 604.176,A -85,B 0,C 180,E1 -29367.124,E2 -29367.124} C_VEL
LIN {X 0,Y 63.931,Z 609.275,A -85,B 0,C 180,E1 -29374.466,E2 -29374.466} C_VEL
LIN {X 0,Y 56.489,Z 612.208,A -85,B 0,C 180,E1 -29381.715,E2 -29381.715} C_VEL
LIN {X 0,Y 48.319,Z 615.066,A -85,B 0,C 180,E1 -29394.424,E2 -29394.424} C_VEL
LIN {X 0,Y 43.049,Z 616.772,A -85,B 0,C 180,E1 -29410.944,E2 -29410.944} C_VEL
LIN {X 0,Y 41.426,Z 617.356,A -85,B 0,C 180,E1 -29430,E2 -29430} C_VEL
LIN {X 0,Y 43.043,Z 616.799,A -85,B 0,C 180,E1 -29449.059,E2 -29449.059} C_VEL
LIN {X 0,Y 48.266,Z 615.131,A -85,B 0,C 180,E1 -29465.621,E2 -29465.621} C_VEL
LIN {X 0,Y 56.464,Z 612.303,A -85,B 0,C 180,E1 -29478.313,E2 -29478.313} C_VEL
LIN {X 0,Y 66.589,Z 608.246,A -85,B 0,C 180,E1 -29487.599,E2 -29487.599} C_VEL
LIN {X 0,Y 77.904,Z 602.862,A -85,B 0,C 180,E1 -29494.437,E2 -29494.437} C_VEL
LIN {X 0,Y 90.039,Z 595.991,A -85,B 0,C 180,E1 -29499.494,E2 -29499.494} C_VEL
LIN {X 0,Y 102.695,Z 587.408,A -85,B 0,C 180,E1 -29503.351,E2 -29503.351} C_VEL
LIN {X 0,Y 110.728,Z 581.043,A -85,B 0,C 180,E1 -29505.445,E2 -29505.445} C_VEL
LIN {X 0,Y 122.275,Z 570.599,A -85,B 0,C 180,E1 -29507.709,E2 -29507.709} C_VEL
LIN {X 0,Y 132.277,Z 559.866,A -85,B 0,C 180,E1 -29509.387,E2 -29509.387} C_VEL
LIN {X 0,Y 141.534,Z 548.142,A -85,B 0,C 180,E1 -29510.71,E2 -29510.71} C_VEL
LIN {X 0,Y 150.034,Z 535.247,A -85,B 0,C 180,E1 -29511.844,E2 -29511.844} C_VEL
LIN {X 0,Y 156.774,Z 522.948,A -85,B 0,C 180,E1 -29512.662,E2 -29512.662} C_VEL
LIN {X 0,Y 162.739,Z 509.635,A -85,B 0,C 180,E1 -29513.336,E2 -29513.336} C_VEL
LIN {X 0,Y 167.948,Z 494.67,A -85,B 0,C 180,E1 -29513.877,E2 -29513.877} C_VEL
LIN {X 0,Y 171.608,Z 480.35,A -85,B 0,C 180,E1 -29514.25,E2 -29514.25} C_VEL
LIN {X 0,Y 174.134,Z 464.988,A -85,B 0,C 180,E1 -29514.572,E2 -29514.572} C_VEL
LIN {X 0,Y 173.793,Z 461.831,A -85,B 0,C 180,E1 -29520,E2 -29520} C_VEL
LIN {X 0,Y 174.111,Z 464.869,A -85,B 0,C 180,E1 -29524.933,E2 -29524.933} C_VEL
LIN {X 0,Y 174.146,Z 465.057,A -85,B 0,C 180,E1 -29525.143,E2 -29525.143} C_VEL
LIN {X 0,Y 171.56,Z 481.005,A -85,B 0,C 180,E1 -29525.417,E2 -29525.417} C_VEL
LIN {X 0,Y 167.481,Z 496.798,A -85,B 0,C 180,E1 -29525.754,E2 -29525.754} C_VEL
LIN {X 0,Y 162.152,Z 511.731,A -85,B 0,C 180,E1 -29526.211,E2 -29526.211} C_VEL
LIN {X 0,Y 155.703,Z 525.77,A -85,B 0,C 180,E1 -29526.789,E2 -29526.789} C_VEL
LIN {X 0,Y 147.992,Z 539.318,A -85,B 0,C 180,E1 -29527.561,E2 -29527.561} C_VEL
LIN {X 0,Y 139.627,Z 551.501,A -85,B 0,C 180,E1 -29528.545,E2 -29528.545} C_VEL
LIN {X 0,Y 130.185,Z 563.131,A -85,B 0,C 180,E1 -29529.871,E2 -29529.871} C_VEL
LIN {X 0,Y 120.085,Z 573.63,A -85,B 0,C 180,E1 -29531.399,E2 -29531.399} C_VEL
LIN {X 0,Y 108.487,Z 583.909,A -85,B 0,C 180,E1 -29533.664,E2 -29533.664} C_VEL
LIN {X 0,Y 97.102,Z 592.458,A -85,B 0,C 180,E1 -29536.469,E2 -29536.469} C_VEL
LIN {X 0,Y 86.097,Z 599.584,A -85,B 0,C 180,E1 -29540.164,E2 -29540.164} C_VEL
LIN {X 0,Y 73.982,Z 606.198,A -85,B 0,C 180,E1 -29545.519,E2 -29545.519} C_VEL
LIN {X 0,Y 62.795,Z 611.383,A -85,B 0,C 180,E1 -29552.926,E2 -29552.926} C_VEL
LIN {X 0,Y 55.351,Z 614.395,A -85,B 0,C 180,E1 -29560.376,E2 -29560.376} C_VEL
LIN {X 0,Y 47.236,Z 617.334,A -85,B 0,C 180,E1 -29573.479,E2 -29573.479} C_VEL
LIN {X 0,Y 42.281,Z 619.1,A -85,B 0,C 180,E1 -29590.583,E2 -29590.583} C_VEL
LIN {X 0,Y 41.264,Z 619.721,A -85,B 0,C 180,E1 -29610,E2 -29610} C_VEL
LIN {X 0,Y 42.271,Z 619.077,A -85,B 0,C 180,E1 -29629.421,E2 -29629.421} C_VEL
LIN {X 0,Y 47.207,Z 617.279,A -85,B 0,C 180,E1 -29646.547,E2 -29646.547} C_VEL
LIN {X 0,Y 55.268,Z 614.312,A -85,B 0,C 180,E1 -29659.725,E2 -29659.725} C_VEL
LIN {X 0,Y 65.493,Z 610.113,A -85,B 0,C 180,E1 -29669.143,E2 -29669.143} C_VEL
LIN {X 0,Y 76.951,Z 604.567,A -85,B 0,C 180,E1 -29675.963,E2 -29675.963} C_VEL
LIN {X 0,Y 89.215,Z 597.527,A -85,B 0,C 180,E1 -29680.959,E2 -29680.959} C_VEL
LIN {X 0,Y 100.325,Z 590.003,A -85,B 0,C 180,E1 -29684.406,E2 -29684.406} C_VEL
LIN {X 0,Y 111.784,Z 580.947,A -85,B 0,C 180,E1 -29687.026,E2 -29687.026} C_VEL
LIN {X 0,Y 121.757,Z 571.705,A -85,B 0,C 180,E1 -29688.884,E2 -29688.884} C_VEL
LIN {X 0,Y 131.858,Z 560.823,A -85,B 0,C 180,E1 -29690.406,E2 -29690.406} C_VEL
LIN {X 0,Y 141.207,Z 548.885,A -85,B 0,C 180,E1 -29691.681,E2 -29691.681} C_VEL
LIN {X 0,Y 149.7,Z 535.952,A -85,B 0,C 180,E1 -29692.626,E2 -29692.626} C_VEL
LIN {X 0,Y 157.418,Z 521.593,A -85,B 0,C 180,E1 -29693.381,E2 -29693.381} C_VEL
LIN {X 0,Y 163.295,Z 507.948,A -85,B 0,C 180,E1 -29693.885,E2 -29693.885} C_VEL
LIN {X 0,Y 168.256,Z 493.002,A -85,B 0,C 180,E1 -29694.308,E2 -29694.308} C_VEL
LIN {X 0,Y 171.928,Z 477.392,A -85,B 0,C 180,E1 -29694.62,E2 -29694.62} C_VEL
LIN {X 0,Y 173.861,Z 464.755,A -85,B 0,C 180,E1 -29694.853,E2 -29694.853} C_VEL
LIN {X 0,Y 173.532,Z 463.255,A -85,B 0,C 180,E1 -29697.144,E2 -29697.144} C_VEL
LIN {X 0,Y 173.376,Z 463.603,A -85,B 0,C 180,E1 -29697.985,E2 -29697.985} C_VEL
LIN {X 0,Y 173.054,Z 465.453,A -85,B 0,C 180,E1 -29698.951,E2 -29698.951} C_VEL
LIN {X 0,Y 172.566,Z 468.535,A -85,B 0,C 180,E1 -29700.377,E2 -29700.377} C_VEL
LIN {X 0,Y 172.514,Z 468.927,A -85,B 0,C 180,E1 -29700.757,E2 -29700.757} C_VEL
LIN {X 0,Y 172.525,Z 470.423,A -85,B 0,C 180,E1 -29703.258,E2 -29703.258} C_VEL
LIN {X 0,Y 169.652,Z 485.061,A -85,B 0,C 180,E1 -29703.558,E2 -29703.558} C_VEL
LIN {X 0,Y 165.806,Z 498.64,A -85,B 0,C 180,E1 -29703.912,E2 -29703.912} C_VEL
LIN {X 0,Y 160.355,Z 513.11,A -85,B 0,C 180,E1 -29704.402,E2 -29704.402} C_VEL
LIN {X 0,Y 154.366,Z 525.764,A -85,B 0,C 180,E1 -29704.985,E2 -29704.985} C_VEL
LIN {X 0,Y 147.44,Z 537.814,A -85,B 0,C 180,E1 -29705.723,E2 -29705.723} C_VEL
LIN {X 0,Y 138.009,Z 551.378,A -85,B 0,C 180,E1 -29706.786,E2 -29706.786} C_VEL
LIN {X 0,Y 127.772,Z 563.534,A -85,B 0,C 180,E1 -29708.092,E2 -29708.092} C_VEL
LIN {X 0,Y 117.589,Z 573.714,A -85,B 0,C 180,E1 -29709.553,E2 -29709.553} C_VEL
LIN {X 0,Y 105.839,Z 583.667,A -85,B 0,C 180,E1 -29711.666,E2 -29711.666} C_VEL
LIN {X 0,Y 95.984,Z 590.79,A -85,B 0,C 180,E1 -29714.035,E2 -29714.035} C_VEL
LIN {X 0,Y 84.613,Z 597.844,A -85,B 0,C 180,E1 -29717.22,E2 -29717.22} C_VEL
LIN {X 0,Y 72.04,Z 604.381,A -85,B 0,C 180,E1 -29722.064,E2 -29722.064} C_VEL
LIN {X 0,Y 60.184,Z 609.48,A -85,B 0,C 180,E1 -29728.862,E2 -29728.862} C_VEL
LIN {X 0,Y 52.011,Z 612.413,A -85,B 0,C 180,E1 -29735.833,E2 -29735.833} C_VEL
LIN {X 0,Y 42.728,Z 615.271,A -85,B 0,C 180,E1 -29748.86,E2 -29748.86} C_VEL
LIN {X 0,Y 36.408,Z 616.975,A -85,B 0,C 180,E1 -29767.29,E2 -29767.29} C_VEL
LIN {X 0,Y 34.328,Z 617.559,A -85,B 0,C 180,E1 -29790,E2 -29790} C_VEL
LIN {X 0,Y 36.401,Z 617.002,A -85,B 0,C 180,E1 -29812.714,E2 -29812.714} C_VEL
LIN {X 0,Y 42.667,Z 615.335,A -85,B 0,C 180,E1 -29831.212,E2 -29831.212} C_VEL
LIN {X 0,Y 51.99,Z 612.507,A -85,B 0,C 180,E1 -29844.2,E2 -29844.2} C_VEL
LIN {X 0,Y 63.045,Z 608.45,A -85,B 0,C 180,E1 -29853.099,E2 -29853.099} C_VEL
LIN {X 0,Y 75.099,Z 603.065,A -85,B 0,C 180,E1 -29859.358,E2 -29859.358} C_VEL
LIN {X 0,Y 87.789,Z 596.194,A -85,B 0,C 180,E1 -29863.872,E2 -29863.872} C_VEL
LIN {X 0,Y 99.244,Z 588.805,A -85,B 0,C 180,E1 -29866.825,E2 -29866.825} C_VEL
LIN {X 0,Y 107.479,Z 582.591,A -85,B 0,C 180,E1 -29868.758,E2 -29868.758} C_VEL
LIN {X 0,Y 119.269,Z 572.419,A -85,B 0,C 180,E1 -29870.742,E2 -29870.742} C_VEL
LIN {X 0,Y 129.453,Z 562.009,A -85,B 0,C 180,E1 -29872.206,E2 -29872.206} C_VEL
LIN {X 0,Y 138.848,Z 550.679,A -85,B 0,C 180,E1 -29873.375,E2 -29873.375} C_VEL
LIN {X 0,Y 147.426,Z 538.366,A -85,B 0,C 180,E1 -29874.333,E2 -29874.333} C_VEL
LIN {X 0,Y 154.217,Z 526.642,A -85,B 0,C 180,E1 -29875.064,E2 -29875.064} C_VEL
LIN {X 0,Y 160.34,Z 513.896,A -85,B 0,C 180,E1 -29875.672,E2 -29875.672} C_VEL
LIN {X 0,Y 166.023,Z 498.959,A -85,B 0,C 180,E1 -29876.173,E2 -29876.173} C_VEL
LIN {X 0,Y 170.351,Z 483.483,A -85,B 0,C 180,E1 -29876.57,E2 -29876.57} C_VEL
LIN {X 0,Y 172.812,Z 470.728,A -85,B 0,C 180,E1 -29876.814,E2 -29876.814} C_VEL
LIN {X 0,Y 172.833,Z 469.003,A -85,B 0,C 180,E1 -29880,E2 -29880} C_VEL
LIN {X 0,Y 172.833,Z 470.706,A -85,B 0,C 180,E1 -29882.866,E2 -29882.866} C_VEL
LIN {X 0,Y 169.93,Z 485.547,A -85,B 0,C 180,E1 -29883.133,E2 -29883.133} C_VEL
LIN {X 0,Y 165.666,Z 500.376,A -85,B 0,C 180,E1 -29883.433,E2 -29883.433} C_VEL
LIN {X 0,Y 160.234,Z 514.525,A -85,B 0,C 180,E1 -29883.797,E2 -29883.797} C_VEL
LIN {X 0,Y 153.288,Z 528.756,A -85,B 0,C 180,E1 -29884.308,E2 -29884.308} C_VEL
LIN {X 0,Y 145.491,Z 541.725,A -85,B 0,C 180,E1 -29884.951,E2 -29884.951} C_VEL
LIN {X 0,Y 136.763,Z 553.852,A -85,B 0,C 180,E1 -29885.844,E2 -29885.844} C_VEL
LIN {X 0,Y 127.436,Z 564.827,A -85,B 0,C 180,E1 -29886.948,E2 -29886.948} C_VEL
LIN {X 0,Y 117.175,Z 575.06,A -85,B 0,C 180,E1 -29888.263,E2 -29888.263} C_VEL
LIN {X 0,Y 105.339,Z 585.064,A -85,B 0,C 180,E1 -29890.243,E2 -29890.243} C_VEL
LIN {X 0,Y 93.668,Z 593.38,A -85,B 0,C 180,E1 -29892.74,E2 -29892.74} C_VEL
LIN {X 0,Y 80.684,Z 601.205,A -85,B 0,C 180,E1 -29896.639,E2 -29896.639} C_VEL
LIN {X 0,Y 68.11,Z 607.432,A -85,B 0,C 180,E1 -29901.774,E2 -29901.774} C_VEL
LIN {X 0,Y 56.378,Z 612.261,A -85,B 0,C 180,E1 -29909.24,E2 -29909.24} C_VEL
LIN {X 0,Y 46.037,Z 615.81,A -85,B 0,C 180,E1 -29920.246,E2 -29920.246} C_VEL
LIN {X 0,Y 38.124,Z 618.155,A -85,B 0,C 180,E1 -29936.425,E2 -29936.425} C_VEL
LIN {X 0,Y 34.259,Z 619.351,A -85,B 0,C 180,E1 -29958.162,E2 -29958.162} C_VEL
LIN {X 0,Y 34.142,Z 619.517,A -85,B 0,C 180,E1 -29970,E2 -29970} C_VEL
LIN {X 0,Y 35.605,Z 618.872,A -85,B 0,C 180,E1 -29993.251,E2 -29993.251} C_VEL
LIN {X 0,Y 41.659,Z 617.074,A -85,B 0,C 180,E1 -30012.438,E2 -30012.438} C_VEL
LIN {X 0,Y 50.922,Z 614.106,A -85,B 0,C 180,E1 -30025.9,E2 -30025.9} C_VEL
LIN {X 0,Y 62.12,Z 609.907,A -85,B 0,C 180,E1 -30034.831,E2 -30034.831} C_VEL
LIN {X 0,Y 74.321,Z 604.361,A -85,B 0,C 180,E1 -30041.015,E2 -30041.015} C_VEL
LIN {X 0,Y 87.142,Z 597.321,A -85,B 0,C 180,E1 -30045.414,E2 -30045.414} C_VEL
LIN {X 0,Y 98.643,Z 589.797,A -85,B 0,C 180,E1 -30048.412,E2 -30048.412} C_VEL
LIN {X 0,Y 110.401,Z 580.741,A -85,B 0,C 180,E1 -30050.639,E2 -30050.639} C_VEL
LIN {X 0,Y 120.585,Z 571.498,A -85,B 0,C 180,E1 -30052.209,E2 -30052.209} C_VEL
LIN {X 0,Y 130.856,Z 560.616,A -85,B 0,C 180,E1 -30053.499,E2 -30053.499} C_VEL
LIN {X 0,Y 140.222,Z 548.852,A -85,B 0,C 180,E1 -30054.555,E2 -30054.555} C_VEL
LIN {X 0,Y 148.955,Z 535.744,A -85,B 0,C 180,E1 -30055.338,E2 -30055.338} C_VEL
LIN {X 0,Y 156.758,Z 521.385,A -85,B 0,C 180,E1 -30055.961,E2 -30055.961} C_VEL
LIN {X 0,Y 162.606,Z 507.959,A -85,B 0,C 180,E1 -30056.37,E2 -30056.37} C_VEL
LIN {X 0,Y 167.621,Z 493.07,A -85,B 0,C 180,E1 -30056.715,E2 -30056.715} C_VEL
LIN {X 0,Y 171.394,Z 477.248,A -85,B 0,C 180,E1 -30056.985,E2 -30056.985} C_VEL
LIN {X 0,Y 172.546,Z 470.441,A -85,B 0,C 180,E1 -30057.12,E2 -30057.12} C_VEL
LIN {X 0,Y 172.556,Z 468.603,A -85,B 0,C 180,E1 -30060,E2 -30060} C_VEL
LIN {X 0,Y 172.514,Z 468.927,A -85,B 0,C 180,E1 -30060.757,E2 -30060.757} C_VEL
LIN {X 0,Y 172.364,Z 470.209,A -85,B 0,C 180,E1 -30061.376,E2 -30061.376} C_VEL
LIN {X 0,Y 172.073,Z 472.299,A -85,B 0,C 180,E1 -30061.739,E2 -30061.739} C_VEL
LIN {X 0,Y 171.385,Z 476.108,A -85,B 0,C 180,E1 -30061.903,E2 -30061.903} C_VEL
LIN {X 0,Y 168.661,Z 488.2,A -85,B 0,C 180,E1 -30061.253,E2 -30061.253} C_VEL
LIN {X 0,Y 168.233,Z 489.737,A -85,B 0,C 180,E1 -30061.267,E2 -30061.267} C_VEL
LIN {X 0,Y 163.338,Z 504.97,A -85,B 0,C 180,E1 -30061.63,E2 -30061.63} C_VEL
LIN {X 0,Y 157.348,Z 519.129,A -85,B 0,C 180,E1 -30062.057,E2 -30062.057} C_VEL
LIN {X 0,Y 149.687,Z 533.465,A -85,B 0,C 180,E1 -30062.691,E2 -30062.691} C_VEL
LIN {X 0,Y 141.691,Z 545.753,A -85,B 0,C 180,E1 -30063.452,E2 -30063.452} C_VEL
LIN {X 0,Y 132.152,Z 557.944,A -85,B 0,C 180,E1 -30064.35,E2 -30064.35} C_VEL
LIN {X 0,Y 121.796,Z 569.05,A -85,B 0,C 180,E1 -30065.529,E2 -30065.529} C_VEL
LIN {X 0,Y 109.76,Z 579.833,A -85,B 0,C 180,E1 -30067.049,E2 -30067.049} C_VEL
LIN {X 0,Y 101.836,Z 585.924,A -85,B 0,C 180,E1 -30068.376,E2 -30068.376} C_VEL
LIN {X 0,Y 92.819,Z 592.104,A -85,B 0,C 180,E1 -30070.169,E2 -30070.169} C_VEL
LIN {X 0,Y 79.474,Z 599.844,A -85,B 0,C 180,E1 -30073.413,E2 -30073.413} C_VEL
LIN {X 0,Y 66.463,Z 605.996,A -85,B 0,C 180,E1 -30077.888,E2 -30077.888} C_VEL
LIN {X 0,Y 54.046,Z 610.735,A -85,B 0,C 180,E1 -30084.461,E2 -30084.461} C_VEL
LIN {X 0,Y 42.631,Z 614.196,A -85,B 0,C 180,E1 -30094.487,E2 -30094.487} C_VEL
LIN {X 0,Y 33.333,Z 616.467,A -85,B 0,C 180,E1 -30110.764,E2 -30110.764} C_VEL
LIN {X 0,Y 27.883,Z 617.612,A -85,B 0,C 180,E1 -30135.401,E2 -30135.401} C_VEL
LIN {X 0,Y 27.245,Z 617.762,A -85,B 0,C 180,E1 -30150,E2 -30150} C_VEL
LIN {X 0,Y 29.958,Z 617.205,A -85,B 0,C 180,E1 -30177.981,E2 -30177.981} C_VEL
LIN {X 0,Y 37.599,Z 615.538,A -85,B 0,C 180,E1 -30198.387,E2 -30198.387} C_VEL
LIN {X 0,Y 48.164,Z 612.71,A -85,B 0,C 180,E1 -30211.101,E2 -30211.101} C_VEL
LIN {X 0,Y 61.739,Z 608.024,A -85,B 0,C 180,E1 -30220.031,E2 -30220.031} C_VEL
LIN {X 0,Y 72.893,Z 603.267,A -85,B 0,C 180,E1 -30224.606,E2 -30224.606} C_VEL
LIN {X 0,Y 86.077,Z 596.397,A -85,B 0,C 180,E1 -30228.45,E2 -30228.45} C_VEL
LIN {X 0,Y 97.862,Z 589.007,A -85,B 0,C 180,E1 -30230.909,E2 -30230.909} C_VEL
LIN {X 0,Y 106.321,Z 582.792,A -85,B 0,C 180,E1 -30232.522,E2 -30232.522} C_VEL
LIN {X 0,Y 118.333,Z 572.62,A -85,B 0,C 180,E1 -30234.146,E2 -30234.146} C_VEL
LIN {X 0,Y 128.681,Z 562.209,A -85,B 0,C 180,E1 -30235.351,E2 -30235.351} C_VEL
LIN {X 0,Y 138.208,Z 550.879,A -85,B 0,C 180,E1 -30236.307,E2 -30236.307} C_VEL
LIN {X 0,Y 147.028,Z 538.352,A -85,B 0,C 180,E1 -30237.11,E2 -30237.11} C_VEL
LIN {X 0,Y 154.727,Z 525.091,A -85,B 0,C 180,E1 -30237.783,E2 -30237.783} C_VEL
LIN {X 0,Y 161.272,Z 511.113,A -85,B 0,C 180,E1 -30238.289,E2 -30238.289} C_VEL
LIN {X 0,Y 166.931,Z 495.408,A -85,B 0,C 180,E1 -30238.714,E2 -30238.714} C_VEL
LIN {X 0,Y 170.933,Z 479.917,A -85,B 0,C 180,E1 -30238.998,E2 -30238.998} C_VEL
LIN {X 0,Y 171.598,Z 476.439,A -85,B 0,C 180,E1 -30239.143,E2 -30239.143} C_VEL
LIN {X 0,Y 171.63,Z 476.262,A -85,B 0,C 180,E1 -30240.173,E2 -30240.173} C_VEL
LIN {X 0,Y 171.601,Z 476.481,A -85,B 0,C 180,E1 -30240.574,E2 -30240.574} C_VEL
LIN {X 0,Y 168.46,Z 490.183,A -85,B 0,C 180,E1 -30240.804,E2 -30240.804} C_VEL
LIN {X 0,Y 164.005,Z 504.227,A -85,B 0,C 180,E1 -30241.051,E2 -30241.051} C_VEL
LIN {X 0,Y 158.17,Z 518.296,A -85,B 0,C 180,E1 -30241.356,E2 -30241.356} C_VEL
LIN {X 0,Y 151.17,Z 531.726,A -85,B 0,C 180,E1 -30241.771,E2 -30241.771} C_VEL
LIN {X 0,Y 142.431,Z 545.404,A -85,B 0,C 180,E1 -30242.336,E2 -30242.336} C_VEL
LIN {X 0,Y 132.88,Z 557.77,A -85,B 0,C 180,E1 -30243.154,E2 -30243.154} C_VEL
LIN {X 0,Y 121.565,Z 569.961,A -85,B 0,C 180,E1 -30244.258,E2 -30244.258} C_VEL
LIN {X 0,Y 111.186,Z 579.351,A -85,B 0,C 180,E1 -30245.423,E2 -30245.423} C_VEL
LIN {X 0,Y 99.162,Z 588.591,A -85,B 0,C 180,E1 -30247.156,E2 -30247.156} C_VEL
LIN {X 0,Y 87.647,Z 596.067,A -85,B 0,C 180,E1 -30249.402,E2 -30249.402} C_VEL
LIN {X 0,Y 75.612,Z 602.675,A -85,B 0,C 180,E1 -30252.598,E2 -30252.598} C_VEL
LIN {X 0,Y 62.579,Z 608.551,A -85,B 0,C 180,E1 -30257.337,E2 -30257.337} C_VEL
LIN {X 0,Y 49.33,Z 613.355,A -85,B 0,C 180,E1 -30265.302,E2 -30265.302} C_VEL
LIN {X 0,Y 36.714,Z 616.924,A -85,B 0,C 180,E1 -30280.032,E2 -30280.032} C_VEL
LIN {X 0,Y 29.182,Z 618.692,A -85,B 0,C 180,E1 -30301.207,E2 -30301.207} C_VEL
LIN {X 0,Y 27.028,Z 619.314,A -85,B 0,C 180,E1 -30330,E2 -30330} C_VEL
LIN {X 0,Y 29.158,Z 618.667,A -85,B 0,C 180,E1 -30358.819,E2 -30358.819} C_VEL
LIN {X 0,Y 36.686,Z 616.868,A -85,B 0,C 180,E1 -30380.019,E2 -30380.019} C_VEL
LIN {X 0,Y 48.963,Z 613.377,A -85,B 0,C 180,E1 -30394.495,E2 -30394.495} C_VEL
LIN {X 0,Y 62.585,Z 608.444,A -85,B 0,C 180,E1 -30402.645,E2 -30402.645} C_VEL
LIN {X 0,Y 75.621,Z 602.528,A -85,B 0,C 180,E1 -30407.373,E2 -30407.373} C_VEL
LIN {X 0,Y 89.388,Z 594.833,A -85,B 0,C 180,E1 -30410.953,E2 -30410.953} C_VEL
LIN {X 0,Y 100.874,Z 587.124,A -85,B 0,C 180,E1 -30413.111,E2 -30413.111} C_VEL
LIN {X 0,Y 112.907,Z 577.584,A -85,B 0,C 180,E1 -30414.812,E2 -30414.812} C_VEL
LIN {X 0,Y 123.297,Z 567.872,A -85,B 0,C 180,E1 -30415.933,E2 -30415.933} C_VEL
LIN {X 0,Y 133.719,Z 556.34,A -85,B 0,C 180,E1 -30416.941,E2 -30416.941} C_VEL
LIN {X 0,Y 143.304,Z 543.639,A -85,B 0,C 180,E1 -30417.728,E2 -30417.728} C_VEL
LIN {X 0,Y 151.168,Z 531.128,A -85,B 0,C 180,E1 -30418.25,E2 -30418.25} C_VEL
LIN {X 0,Y 158.169,Z 517.553,A -85,B 0,C 180,E1 -30418.649,E2 -30418.649} C_VEL
LIN {X 0,Y 164.206,Z 502.732,A -85,B 0,C 180,E1 -30418.98,E2 -30418.98} C_VEL
LIN {X 0,Y 168.683,Z 488.193,A -85,B 0,C 180,E1 -30419.224,E2 -30419.224} C_VEL
LIN {X 0,Y 171.326,Z 476.188,A -85,B 0,C 180,E1 -30419.415,E2 -30419.415} C_VEL
LIN {X 0,Y 171.379,Z 475.814,A -85,B 0,C 180,E1 -30420,E2 -30420} C_VEL
LIN {X 0,Y 171.309,Z 476.221,A -85,B 0,C 180,E1 -30420.998,E2 -30420.998} C_VEL
LIN {X 0,Y 168.233,Z 489.737,A -85,B 0,C 180,E1 -30421.267,E2 -30421.267} C_VEL
LIN {X 0,Y 168.152,Z 490.31,A -85,B 0,C 180,E1 -30421.275,E2 -30421.275} C_VEL
LIN {X 0,Y 168.152,Z 558.971,A -85,B 0,C 180,E1 -30421.275,E2 -30421.275} C_VEL
LIN {X 0,Y 146.11,Z 558.971,A -85,B 0,C 180,E1 -30420.515,E2 -30420.515} C_VEL
LIN {X 0,Y 144.121,Z 556.971,A -85,B 0,C 180,E1 -30420.435,E2 -30420.435} C_VEL
LIN {X 0,Y 144.121,Z 548.337,A -85,B 0,C 180,E1 -30420.435,E2 -30420.435} C_VEL
LIN {X 0,Y 140.565,Z 547.128,A -85,B 0,C 180,E1 -30420.644,E2 -30420.644} C_VEL
LIN {X 0,Y 131.806,Z 558.148,A -85,B 0,C 180,E1 -30421.265,E2 -30421.265} C_VEL
LIN {X 0,Y 121.317,Z 569.256,A -85,B 0,C 180,E1 -30422.18,E2 -30422.18} C_VEL
